LIN {X 0,Y 467.598,Z 337.24,A -85,B 0,C 180,E1 -7780.262,E2 -7780.262} C_VEL
LIN {X 0,Y 467.588,Z 337.241,A -85,B 0,C 180,E1 -7782.567,E2 -7782.567} C_VEL
LIN {X 0,Y 467.573,Z 337.242,A -85,B 0,C 180,E1 -7785.053,E2 -7785.053} C_VEL
LIN {X 0,Y 467.59,Z 337.241,A -85,B 0,C 180,E1 -7787.44,E2 -7787.44} C_VEL
LIN {X 0,Y 467.584,Z 337.244,A -85,B 0,C 180,E1 -7790.855,E2 -7790.855} C_VEL
LIN {X 0,Y 467.561,Z 337.244,A -85,B 0,C 180,E1 -7794.261,E2 -7794.261} C_VEL
LIN {X 0,Y 467.583,Z 337.239,A -85,B 0,C 180,E1 -7797.321,E2 -7797.321} C_VEL
LIN {X 0,Y 467.571,Z 337.241,A -85,B 0,C 180,E1 -7800.667,E2 -7800.667} C_VEL
LIN {X 0,Y 467.618,Z 337.238,A -85,B 0,C 180,E1 -7803.2,E2 -7803.2} C_VEL
LIN {X 0,Y 467.594,Z 337.24,A -85,B 0,C 180,E1 -7806.468,E2 -7806.468} C_VEL
LIN {X 0,Y 467.625,Z 337.233,A -85,B 0,C 180,E1 -7809.777,E2 -7809.777} C_VEL
LIN {X 0,Y 467.591,Z 337.238,A -85,B 0,C 180,E1 -7812.902,E2 -7812.902} C_VEL
LIN {X 0,Y 466.915,Z 337.324,A -85,B 0,C 180,E1 -7813.621,E2 -7813.621} C_VEL
LIN {X 0,Y 464.043,Z 337.68,A -85,B 0,C 180,E1 -7814.788,E2 -7814.788} C_VEL
LIN {X 0,Y 461.631,Z 337.984,A -85,B 0,C 180,E1 -7815.729,E2 -7815.729} C_VEL
LIN {X 0,Y 460.615,Z 338.108,A -85,B 0,C 180,E1 -7816.456,E2 -7816.456} C_VEL
LIN {X 0,Y 460.543,Z 338.117,A -85,B 0,C 180,E1 -7816.703,E2 -7816.703} C_VEL
LIN {X 0,Y 460.581,Z 338.114,A -85,B 0,C 180,E1 -7819.449,E2 -7819.449} C_VEL
LIN {X 0,Y 460.716,Z 338.099,A -85,B 0,C 180,E1 -7822.543,E2 -7822.543} C_VEL
LIN {X 0,Y 460.697,Z 338.099,A -85,B 0,C 180,E1 -7824.748,E2 -7824.748} C_VEL
LIN {X 0,Y 460.826,Z 338.08,A -85,B 0,C 180,E1 -7827.378,E2 -7827.378} C_VEL
LIN {X 0,Y 460.854,Z 338.082,A -85,B 0,C 180,E1 -7830,E2 -7830} C_VEL
LIN {X 0,Y 460.827,Z 338.081,A -85,B 0,C 180,E1 -7832.622,E2 -7832.622} C_VEL
LIN {X 0,Y 460.704,Z 338.097,A -85,B 0,C 180,E1 -7836.13,E2 -7836.13} C_VEL
LIN {X 0,Y 460.631,Z 338.108,A -85,B 0,C 180,E1 -7838.776,E2 -7838.776} C_VEL
LIN {X 0,Y 460.615,Z 338.109,A -85,B 0,C 180,E1 -7842.445,E2 -7842.445} C_VEL
LIN {X 0,Y 460.601,Z 338.111,A -85,B 0,C 180,E1 -7845.998,E2 -7845.998} C_VEL
LIN {X 0,Y 460.573,Z 338.113,A -85,B 0,C 180,E1 -7848.902,E2 -7848.902} C_VEL
LIN {X 0,Y 460.517,Z 338.122,A -85,B 0,C 180,E1 -7851.486,E2 -7851.486} C_VEL
LIN {X 0,Y 460.543,Z 338.119,A -85,B 0,C 180,E1 -7854.332,E2 -7854.332} C_VEL
LIN {X 0,Y 460.575,Z 338.113,A -85,B 0,C 180,E1 -7857.244,E2 -7857.244} C_VEL
LIN {X 0,Y 460.512,Z 338.121,A -85,B 0,C 180,E1 -7860.24,E2 -7860.24} C_VEL
LIN {X 0,Y 460.531,Z 338.121,A -85,B 0,C 180,E1 -7863.325,E2 -7863.325} C_VEL
LIN {X 0,Y 460.478,Z 338.124,A -85,B 0,C 180,E1 -7866.53,E2 -7866.53} C_VEL
LIN {X 0,Y 460.535,Z 338.118,A -85,B 0,C 180,E1 -7869.863,E2 -7869.863} C_VEL
LIN {X 0,Y 460.545,Z 338.118,A -85,B 0,C 180,E1 -7872.905,E2 -7872.905} C_VEL
LIN {X 0,Y 460.514,Z 338.123,A -85,B 0,C 180,E1 -7875.831,E2 -7875.831} C_VEL
LIN {X 0,Y 460.534,Z 338.119,A -85,B 0,C 180,E1 -7878.989,E2 -7878.989} C_VEL
LIN {X 0,Y 460.529,Z 338.122,A -85,B 0,C 180,E1 -7881.267,E2 -7881.267} C_VEL
LIN {X 0,Y 460.514,Z 338.121,A -85,B 0,C 180,E1 -7884.555,E2 -7884.555} C_VEL
LIN {X 0,Y 460.535,Z 338.119,A -85,B 0,C 180,E1 -7887.716,E2 -7887.716} C_VEL
LIN {X 0,Y 460.544,Z 338.117,A -85,B 0,C 180,E1 -7890.769,E2 -7890.769} C_VEL
LIN {X 0,Y 460.568,Z 338.115,A -85,B 0,C 180,E1 -7893.735,E2 -7893.735} C_VEL
LIN {X 0,Y 460.55,Z 338.116,A -85,B 0,C 180,E1 -7896.624,E2 -7896.624} C_VEL
LIN {X 0,Y 460.555,Z 338.114,A -85,B 0,C 180,E1 -7899.453,E2 -7899.453} C_VEL
LIN {X 0,Y 460.562,Z 338.115,A -85,B 0,C 180,E1 -7902.23,E2 -7902.23} C_VEL
LIN {X 0,Y 460.571,Z 338.114,A -85,B 0,C 180,E1 -7904.965,E2 -7904.965} C_VEL
LIN {X 0,Y 460.617,Z 338.108,A -85,B 0,C 180,E1 -7908.56,E2 -7908.56} C_VEL
LIN {X 0,Y 460.701,Z 338.097,A -85,B 0,C 180,E1 -7912.109,E2 -7912.109} C_VEL
LIN {X 0,Y 460.701,Z 338.102,A -85,B 0,C 180,E1 -7914.748,E2 -7914.748} C_VEL
LIN {X 0,Y 460.804,Z 338.082,A -85,B 0,C 180,E1 -7917.378,E2 -7917.378} C_VEL
LIN {X 0,Y 460.859,Z 338.079,A -85,B 0,C 180,E1 -7920,E2 -7920} C_VEL
LIN {X 0,Y 460.83,Z 338.081,A -85,B 0,C 180,E1 -7922.622,E2 -7922.622} C_VEL
LIN {X 0,Y 460.705,Z 338.098,A -85,B 0,C 180,E1 -7926.13,E2 -7926.13} C_VEL
LIN {X 0,Y 460.625,Z 338.11,A -85,B 0,C 180,E1 -7928.776,E2 -7928.776} C_VEL
LIN {X 0,Y 460.619,Z 338.112,A -85,B 0,C 180,E1 -7932.445,E2 -7932.445} C_VEL
LIN {X 0,Y 460.606,Z 338.112,A -85,B 0,C 180,E1 -7935.998,E2 -7935.998} C_VEL
LIN {X 0,Y 460.577,Z 338.112,A -85,B 0,C 180,E1 -7938.902,E2 -7938.902} C_VEL
LIN {X 0,Y 460.521,Z 338.122,A -85,B 0,C 180,E1 -7941.486,E2 -7941.486} C_VEL
LIN {X 0,Y 460.547,Z 338.117,A -85,B 0,C 180,E1 -7944.332,E2 -7944.332} C_VEL
LIN {X 0,Y 460.578,Z 338.113,A -85,B 0,C 180,E1 -7947.244,E2 -7947.244} C_VEL
LIN {X 0,Y 460.516,Z 338.124,A -85,B 0,C 180,E1 -7950.24,E2 -7950.24} C_VEL
LIN {X 0,Y 460.534,Z 338.117,A -85,B 0,C 180,E1 -7953.325,E2 -7953.325} C_VEL
LIN {X 0,Y 460.483,Z 338.124,A -85,B 0,C 180,E1 -7956.529,E2 -7956.529} C_VEL
LIN {X 0,Y 460.55,Z 338.117,A -85,B 0,C 180,E1 -7958.898,E2 -7958.898} C_VEL
LIN {X 0,Y 460.527,Z 338.121,A -85,B 0,C 180,E1 -7962.181,E2 -7962.181} C_VEL
LIN {X 0,Y 460.525,Z 338.12,A -85,B 0,C 180,E1 -7965.412,E2 -7965.412} C_VEL
LIN {X 0,Y 460.571,Z 338.31,A -85,B 0,C 180,E1 -7968.756,E2 -7968.756} C_VEL
LIN {X 0,Y 462.718,Z 348.896,A -85,B 0,C 180,E1 -7971.857,E2 -7971.857} C_VEL
LIN {X 0,Y 463.646,Z 354.59,A -85,B 0,C 180,E1 -7973.454,E2 -7973.454} C_VEL
LIN {X 0,Y 463.132,Z 363.771,A -85,B 0,C 180,E1 -7975.842,E2 -7975.842} C_VEL
LIN {X 0,Y 462.412,Z 376.769,A -85,B 0,C 180,E1 -7979.139,E2 -7979.139} C_VEL
LIN {X 0,Y 461.808,Z 389.925,A -85,B 0,C 180,E1 -7982.39,E2 -7982.39} C_VEL
LIN {X 0,Y 461.251,Z 403.652,A -85,B 0,C 180,E1 -7985.707,E2 -7985.707} C_VEL
LIN {X 0,Y 460.785,Z 417.545,A -85,B 0,C 180,E1 -7988.996,E2 -7988.996} C_VEL
LIN {X 0,Y 460.418,Z 431.373,A -85,B 0,C 180,E1 -7992.224,E2 -7992.224} C_VEL
LIN {X 0,Y 460.213,Z 440.731,A -85,B 0,C 180,E1 -7994.39,E2 -7994.39} C_VEL
LIN {X 0,Y 461.598,Z 455.243,A -85,B 0,C 180,E1 -7994.821,E2 -7994.821} C_VEL
LIN {X 0,Y 462.615,Z 466.865,A -85,B 0,C 180,E1 -7995.314,E2 -7995.314} C_VEL
LIN {X 0,Y 462.114,Z 478.343,A -85,B 0,C 180,E1 -7995.916,E2 -7995.916} C_VEL
LIN {X 0,Y 461.604,Z 489.684,A -85,B 0,C 180,E1 -7996.686,E2 -7996.686} C_VEL
LIN {X 0,Y 461.147,Z 501.298,A -85,B 0,C 180,E1 -7997.68,E2 -7997.68} C_VEL
LIN {X 0,Y 460.644,Z 511.654,A -85,B 0,C 180,E1 -7998.783,E2 -7998.783} C_VEL
LIN {X 0,Y 460.277,Z 520.097,A -85,B 0,C 180,E1 -7999.887,E2 -7999.887} C_VEL
LIN {X 0,Y 460.023,Z 528.384,A -85,B 0,C 180,E1 -8001.212,E2 -8001.212} C_VEL
LIN {X 0,Y 459.932,Z 535.07,A -85,B 0,C 180,E1 -8002.537,E2 -8002.537} C_VEL
LIN {X 0,Y 459.913,Z 540.386,A -85,B 0,C 180,E1 -8003.859,E2 -8003.859} C_VEL
LIN {X 0,Y 459.893,Z 544.486,A -85,B 0,C 180,E1 -8005.179,E2 -8005.179} C_VEL
LIN {X 0,Y 459.918,Z 547.493,A -85,B 0,C 180,E1 -8006.496,E2 -8006.496} C_VEL
LIN {X 0,Y 459.904,Z 548.924,A -85,B 0,C 180,E1 -8007.372,E2 -8007.372} C_VEL
LIN {X 0,Y 459.897,Z 549.91,A -85,B 0,C 180,E1 -8008.249,E2 -8008.249} C_VEL
LIN {X 0,Y 460.04,Z 550.668,A -85,B 0,C 180,E1 -8010,E2 -8010} C_VEL
LIN {X 0,Y 460.058,Z 550.379,A -85,B 0,C 180,E1 -8010.875,E2 -8010.875} C_VEL
LIN {X 0,Y 459.953,Z 548.51,A -85,B 0,C 180,E1 -8012.627,E2 -8012.627} C_VEL
LIN {X 0,Y 460.005,Z 545.972,A -85,B 0,C 180,E1 -8013.942,E2 -8013.942} C_VEL
LIN {X 0,Y 459.99,Z 542.372,A -85,B 0,C 180,E1 -8015.26,E2 -8015.26} C_VEL
LIN {X 0,Y 459.99,Z 537.034,A -85,B 0,C 180,E1 -8016.729,E2 -8016.729} C_VEL
LIN {X 0,Y 460.043,Z 530.486,A -85,B 0,C 180,E1 -8018.124,E2 -8018.124} C_VEL
LIN {X 0,Y 460.195,Z 522.709,A -85,B 0,C 180,E1 -8019.449,E2 -8019.449} C_VEL
LIN {X 0,Y 460.5,Z 513.145,A -85,B 0,C 180,E1 -8020.775,E2 -8020.775} C_VEL
LIN {X 0,Y 460.903,Z 503.312,A -85,B 0,C 180,E1 -8021.879,E2 -8021.879} C_VEL
LIN {X 0,Y 461.223,Z 493.086,A -85,B 0,C 180,E1 -8022.826,E2 -8022.826} C_VEL
LIN {X 0,Y 461.773,Z 480.667,A -85,B 0,C 180,E1 -8023.757,E2 -8023.757} C_VEL
LIN {X 0,Y 462.365,Z 467.344,A -85,B 0,C 180,E1 -8024.525,E2 -8024.525} C_VEL
LIN {X 0,Y 461.97,Z 461.418,A -85,B 0,C 180,E1 -8024.819,E2 -8024.819} C_VEL
LIN {X 0,Y 461.138,Z 447.636,A -85,B 0,C 180,E1 -8025.371,E2 -8025.371} C_VEL
LIN {X 0,Y 460.184,Z 436.063,A -85,B 0,C 180,E1 -8025.707,E2 -8025.707} C_VEL
LIN {X 0,Y 460.345,Z 423.4,A -85,B 0,C 180,E1 -8028.469,E2 -8028.469} C_VEL
LIN {X 0,Y 460.504,Z 409.727,A -85,B 0,C 180,E1 -8031.486,E2 -8031.486} C_VEL
LIN {X 0,Y 460.723,Z 396.07,A -85,B 0,C 180,E1 -8034.562,E2 -8034.562} C_VEL
LIN {X 0,Y 461.007,Z 383.272,A -85,B 0,C 180,E1 -8037.534,E2 -8037.534} C_VEL
LIN {X 0,Y 461.36,Z 370.292,A -85,B 0,C 180,E1 -8040.685,E2 -8040.685} C_VEL
LIN {X 0,Y 461.759,Z 360.404,A -85,B 0,C 180,E1 -8043.225,E2 -8043.225} C_VEL
LIN {X 0,Y 462.522,Z 350.975,A -85,B 0,C 180,E1 -8045.804,E2 -8045.804} C_VEL
LIN {X 0,Y 462.353,Z 347.344,A -85,B 0,C 180,E1 -8046.9,E2 -8046.9} C_VEL
LIN {X 0,Y 460.967,Z 340.192,A -85,B 0,C 180,E1 -8049.354,E2 -8049.354} C_VEL
LIN {X 0,Y 460.548,Z 338.121,A -85,B 0,C 180,E1 -8050.196,E2 -8050.196} C_VEL
LIN {X 0,Y 460.504,Z 338.125,A -85,B 0,C 180,E1 -8053.375,E2 -8053.375} C_VEL
LIN {X 0,Y 460.504,Z 338.123,A -85,B 0,C 180,E1 -8056.625,E2 -8056.625} C_VEL
LIN {X 0,Y 460.545,Z 338.118,A -85,B 0,C 180,E1 -8059.731,E2 -8059.731} C_VEL
LIN {X 0,Y 460.531,Z 338.119,A -85,B 0,C 180,E1 -8062.519,E2 -8062.519} C_VEL
LIN {X 0,Y 460.552,Z 338.118,A -85,B 0,C 180,E1 -8065.624,E2 -8065.624} C_VEL
LIN {X 0,Y 460.541,Z 338.118,A -85,B 0,C 180,E1 -8068.745,E2 -8068.745} C_VEL
LIN {X 0,Y 460.586,Z 338.112,A -85,B 0,C 180,E1 -8072.254,E2 -8072.254} C_VEL
LIN {X 0,Y 460.544,Z 338.118,A -85,B 0,C 180,E1 -8074.704,E2 -8074.704} C_VEL
LIN {X 0,Y 460.515,Z 338.123,A -85,B 0,C 180,E1 -8077.571,E2 -8077.571} C_VEL
LIN {X 0,Y 460.573,Z 338.117,A -85,B 0,C 180,E1 -8080.385,E2 -8080.385} C_VEL
LIN {X 0,Y 460.569,Z 338.116,A -85,B 0,C 180,E1 -8083.146,E2 -8083.146} C_VEL
LIN {X 0,Y 460.633,Z 338.213,A -85,B 0,C 180,E1 -8084.134,E2 -8084.134} C_VEL
LIN {X 0,Y 463.679,Z 348.826,A -85,B 0,C 180,E1 -8084.843,E2 -8084.843} C_VEL
LIN {X 0,Y 463.301,Z 360.273,A -85,B 0,C 180,E1 -8085.617,E2 -8085.617} C_VEL
LIN {X 0,Y 462.89,Z 371.591,A -85,B 0,C 180,E1 -8086.594,E2 -8086.594} C_VEL
LIN {X 0,Y 462.45,Z 380.084,A -85,B 0,C 180,E1 -8087.493,E2 -8087.493} C_VEL
LIN {X 0,Y 461.951,Z 388.673,A -85,B 0,C 180,E1 -8088.593,E2 -8088.593} C_VEL
LIN {X 0,Y 461.543,Z 397.068,A -85,B 0,C 180,E1 -8089.915,E2 -8089.915} C_VEL
LIN {X 0,Y 461.19,Z 403.729,A -85,B 0,C 180,E1 -8091.234,E2 -8091.234} C_VEL
LIN {X 0,Y 460.817,Z 409.881,A -85,B 0,C 180,E1 -8092.801,E2 -8092.801} C_VEL
LIN {X 0,Y 460.572,Z 414.264,A -85,B 0,C 180,E1 -8094.308,E2 -8094.308} C_VEL
LIN {X 0,Y 460.387,Z 416.971,A -85,B 0,C 180,E1 -8095.622,E2 -8095.622} C_VEL
LIN {X 0,Y 460.314,Z 418.215,A -85,B 0,C 180,E1 -8096.499,E2 -8096.499} C_VEL
LIN {X 0,Y 460.232,Z 419.525,A -85,B 0,C 180,E1 -8098.25,E2 -8098.25} C_VEL
LIN {X 0,Y 460.185,Z 419.587,A -85,B 0,C 180,E1 -8099.125,E2 -8099.125} C_VEL
LIN {X 0,Y 460.162,Z 418.481,A -85,B 0,C 180,E1 -8100.875,E2 -8100.875} C_VEL
LIN {X 0,Y 460.236,Z 417.34,A -85,B 0,C 180,E1 -8101.75,E2 -8101.75} C_VEL
LIN {X 0,Y 460.28,Z 414.837,A -85,B 0,C 180,E1 -8103.063,E2 -8103.063} C_VEL
LIN {X 0,Y 460.423,Z 411.338,A -85,B 0,C 180,E1 -8104.377,E2 -8104.377} C_VEL
LIN {X 0,Y 460.603,Z 406.758,A -85,B 0,C 180,E1 -8105.692,E2 -8105.692} C_VEL
LIN {X 0,Y 461.037,Z 399.83,A -85,B 0,C 180,E1 -8107.222,E2 -8107.222} C_VEL
LIN {X 0,Y 461.343,Z 392.328,A -85,B 0,C 180,E1 -8108.542,E2 -8108.542} C_VEL
LIN {X 0,Y 461.654,Z 384.704,A -85,B 0,C 180,E1 -8109.64,E2 -8109.64} C_VEL
LIN {X 0,Y 462.091,Z 375.474,A -85,B 0,C 180,E1 -8110.738,E2 -8110.738} C_VEL
LIN {X 0,Y 462.52,Z 365.237,A -85,B 0,C 180,E1 -8111.726,E2 -8111.726} C_VEL
LIN {X 0,Y 462.763,Z 356.364,A -85,B 0,C 180,E1 -8112.439,E2 -8112.439} C_VEL
LIN {X 0,Y 463.121,Z 347.588,A -85,B 0,C 180,E1 -8113.023,E2 -8113.023} C_VEL
LIN {X 0,Y 460.601,Z 338.114,A -85,B 0,C 180,E1 -8113.635,E2 -8113.635} C_VEL
LIN {X 0,Y 460.562,Z 338.114,A -85,B 0,C 180,E1 -8116.854,E2 -8116.854} C_VEL
LIN {X 0,Y 460.571,Z 338.113,A -85,B 0,C 180,E1 -8119.615,E2 -8119.615} C_VEL
LIN {X 0,Y 460.515,Z 338.121,A -85,B 0,C 180,E1 -8122.428,E2 -8122.428} C_VEL
LIN {X 0,Y 460.571,Z 338.115,A -85,B 0,C 180,E1 -8125.802,E2 -8125.802} C_VEL
LIN {X 0,Y 460.559,Z 338.117,A -85,B 0,C 180,E1 -8128.232,E2 -8128.232} C_VEL
LIN {X 0,Y 460.525,Z 338.123,A -85,B 0,C 180,E1 -8131.283,E2 -8131.283} C_VEL
LIN {X 0,Y 460.535,Z 338.118,A -85,B 0,C 180,E1 -8134.505,E2 -8134.505} C_VEL
LIN {X 0,Y 460.531,Z 338.117,A -85,B 0,C 180,E1 -8137.62,E2 -8137.62} C_VEL
LIN {X 0,Y 460.561,Z 338.117,A -85,B 0,C 180,E1 -8140.272,E2 -8140.272} C_VEL
LIN {X 0,Y 460.502,Z 338.124,A -85,B 0,C 180,E1 -8143.375,E2 -8143.375} C_VEL
LIN {X 0,Y 460.515,Z 338.121,A -85,B 0,C 180,E1 -8146.626,E2 -8146.626} C_VEL
LIN {X 0,Y 460.544,Z 338.117,A -85,B 0,C 180,E1 -8149.73,E2 -8149.73} C_VEL
LIN {X 0,Y 460.501,Z 338.125,A -85,B 0,C 180,E1 -8152.524,E2 -8152.524} C_VEL
LIN {X 0,Y 460.547,Z 338.115,A -85,B 0,C 180,E1 -8155.624,E2 -8155.624} C_VEL
LIN {X 0,Y 460.538,Z 338.118,A -85,B 0,C 180,E1 -8158.744,E2 -8158.744} C_VEL
LIN {X 0,Y 460.59,Z 338.112,A -85,B 0,C 180,E1 -8162.252,E2 -8162.252} C_VEL
LIN {X 0,Y 460.56,Z 338.117,A -85,B 0,C 180,E1 -8164.705,E2 -8164.705} C_VEL
LIN {X 0,Y 460.513,Z 338.12,A -85,B 0,C 180,E1 -8167.571,E2 -8167.571} C_VEL
LIN {X 0,Y 460.571,Z 338.118,A -85,B 0,C 180,E1 -8170.384,E2 -8170.384} C_VEL
LIN {X 0,Y 460.567,Z 338.112,A -85,B 0,C 180,E1 -8173.146,E2 -8173.146} C_VEL
LIN {X 0,Y 460.557,Z 338.119,A -85,B 0,C 180,E1 -8175.868,E2 -8175.868} C_VEL
LIN {X 0,Y 460.543,Z 338.117,A -85,B 0,C 180,E1 -8176.703,E2 -8176.703} C_VEL
LIN {X 0,Y 459.907,Z 338.198,A -85,B 0,C 180,E1 -8177.433,E2 -8177.433} C_VEL
LIN {X 0,Y 457.078,Z 338.55,A -85,B 0,C 180,E1 -8178.62,E2 -8178.62} C_VEL
LIN {X 0,Y 454.674,Z 338.851,A -85,B 0,C 180,E1 -8179.576,E2 -8179.576} C_VEL
LIN {X 0,Y 453.648,Z 338.976,A -85,B 0,C 180,E1 -8180.316,E2 -8180.316} C_VEL
LIN {X 0,Y 453.569,Z 338.985,A -85,B 0,C 180,E1 -8180.566,E2 -8180.566} C_VEL
LIN {X 0,Y 453.631,Z 338.979,A -85,B 0,C 180,E1 -8182.88,E2 -8182.88} C_VEL
LIN {X 0,Y 453.67,Z 338.975,A -85,B 0,C 180,E1 -8184.667,E2 -8184.667} C_VEL
LIN {X 0,Y 453.766,Z 338.96,A -85,B 0,C 180,E1 -8187.337,E2 -8187.337} C_VEL
LIN {X 0,Y 453.824,Z 338.958,A -85,B 0,C 180,E1 -8190,E2 -8190} C_VEL
LIN {X 0,Y 453.767,Z 338.96,A -85,B 0,C 180,E1 -8192.663,E2 -8192.663} C_VEL
LIN {X 0,Y 453.671,Z 338.973,A -85,B 0,C 180,E1 -8196.225,E2 -8196.225} C_VEL
LIN {X 0,Y 453.594,Z 338.984,A -85,B 0,C 180,E1 -8198.913,E2 -8198.913} C_VEL
LIN {X 0,Y 453.565,Z 338.987,A -85,B 0,C 180,E1 -8202.529,E2 -8202.529} C_VEL
LIN {X 0,Y 453.546,Z 338.988,A -85,B 0,C 180,E1 -8206.196,E2 -8206.196} C_VEL
LIN {X 0,Y 453.522,Z 338.991,A -85,B 0,C 180,E1 -8209.041,E2 -8209.041} C_VEL
LIN {X 0,Y 453.478,Z 338.997,A -85,B 0,C 180,E1 -8211.836,E2 -8211.836} C_VEL
LIN {X 0,Y 453.515,Z 338.994,A -85,B 0,C 180,E1 -8214.735,E2 -8214.735} C_VEL
LIN {X 0,Y 453.534,Z 338.994,A -85,B 0,C 180,E1 -8217.96,E2 -8217.96} C_VEL
LIN {X 0,Y 453.468,Z 339.001,A -85,B 0,C 180,E1 -8221.526,E2 -8221.526} C_VEL
LIN {X 0,Y 453.489,Z 338.994,A -85,B 0,C 180,E1 -8224.778,E2 -8224.778} C_VEL
LIN {X 0,Y 453.467,Z 338.999,A -85,B 0,C 180,E1 -8228.312,E2 -8228.312} C_VEL
LIN {X 0,Y 453.497,Z 338.996,A -85,B 0,C 180,E1 -8230.609,E2 -8230.609} C_VEL
LIN {X 0,Y 453.485,Z 338.997,A -85,B 0,C 180,E1 -8233.248,E2 -8233.248} C_VEL
LIN {X 0,Y 453.469,Z 339.001,A -85,B 0,C 180,E1 -8235.779,E2 -8235.779} C_VEL
LIN {X 0,Y 453.482,Z 338.996,A -85,B 0,C 180,E1 -8238.21,E2 -8238.21} C_VEL
LIN {X 0,Y 453.497,Z 338.995,A -85,B 0,C 180,E1 -8240.794,E2 -8240.794} C_VEL
LIN {X 0,Y 453.458,Z 338.998,A -85,B 0,C 180,E1 -8243.918,E2 -8243.918} C_VEL
LIN {X 0,Y 453.486,Z 338.997,A -85,B 0,C 180,E1 -8247.152,E2 -8247.152} C_VEL
LIN {X 0,Y 453.479,Z 338.999,A -85,B 0,C 180,E1 -8250.269,E2 -8250.269} C_VEL
LIN {X 0,Y 453.514,Z 338.996,A -85,B 0,C 180,E1 -8253.295,E2 -8253.295} C_VEL
LIN {X 0,Y 453.507,Z 338.993,A -85,B 0,C 180,E1 -8256.239,E2 -8256.239} C_VEL
LIN {X 0,Y 453.487,Z 338.997,A -85,B 0,C 180,E1 -8259.118,E2 -8259.118} C_VEL
LIN {X 0,Y 453.515,Z 338.992,A -85,B 0,C 180,E1 -8261.945,E2 -8261.945} C_VEL
LIN {X 0,Y 453.545,Z 338.99,A -85,B 0,C 180,E1 -8264.727,E2 -8264.727} C_VEL
LIN {X 0,Y 453.565,Z 338.987,A -85,B 0,C 180,E1 -8268.379,E2 -8268.379} C_VEL
LIN {X 0,Y 453.658,Z 338.975,A -85,B 0,C 180,E1 -8271.985,E2 -8271.985} C_VEL
LIN {X 0,Y 453.675,Z 338.976,A -85,B 0,C 180,E1 -8274.667,E2 -8274.667} C_VEL
LIN {X 0,Y 453.748,Z 338.961,A -85,B 0,C 180,E1 -8277.337,E2 -8277.337} C_VEL
LIN {X 0,Y 453.829,Z 338.954,A -85,B 0,C 180,E1 -8280,E2 -8280} C_VEL
LIN {X 0,Y 453.77,Z 338.961,A -85,B 0,C 180,E1 -8282.663,E2 -8282.663} C_VEL
LIN {X 0,Y 453.672,Z 338.973,A -85,B 0,C 180,E1 -8286.226,E2 -8286.226} C_VEL
LIN {X 0,Y 453.591,Z 338.985,A -85,B 0,C 180,E1 -8288.914,E2 -8288.914} C_VEL
LIN {X 0,Y 453.569,Z 338.989,A -85,B 0,C 180,E1 -8292.529,E2 -8292.529} C_VEL
LIN {X 0,Y 453.55,Z 338.992,A -85,B 0,C 180,E1 -8296.196,E2 -8296.196} C_VEL
LIN {X 0,Y 453.527,Z 338.991,A -85,B 0,C 180,E1 -8299.041,E2 -8299.041} C_VEL
LIN {X 0,Y 453.482,Z 338.999,A -85,B 0,C 180,E1 -8301.836,E2 -8301.836} C_VEL
LIN {X 0,Y 453.519,Z 338.994,A -85,B 0,C 180,E1 -8304.734,E2 -8304.734} C_VEL
LIN {X 0,Y 453.537,Z 338.991,A -85,B 0,C 180,E1 -8307.96,E2 -8307.96} C_VEL
LIN {X 0,Y 453.471,Z 338.997,A -85,B 0,C 180,E1 -8311.525,E2 -8311.525} C_VEL
LIN {X 0,Y 453.494,Z 338.994,A -85,B 0,C 180,E1 -8314.777,E2 -8314.777} C_VEL
LIN {X 0,Y 453.478,Z 338.997,A -85,B 0,C 180,E1 -8318.311,E2 -8318.311} C_VEL
LIN {X 0,Y 453.498,Z 338.996,A -85,B 0,C 180,E1 -8320.609,E2 -8320.609} C_VEL
LIN {X 0,Y 453.46,Z 339,A -85,B 0,C 180,E1 -8323.244,E2 -8323.244} C_VEL
LIN {X 0,Y 453.478,Z 339,A -85,B 0,C 180,E1 -8325.78,E2 -8325.78} C_VEL
LIN {X 0,Y 453.527,Z 339.118,A -85,B 0,C 180,E1 -8328.447,E2 -8328.447} C_VEL
LIN {X 0,Y 455.452,Z 348.745,A -85,B 0,C 180,E1 -8331.322,E2 -8331.322} C_VEL
LIN {X 0,Y 456.645,Z 355.141,A -85,B 0,C 180,E1 -8333.16,E2 -8333.16} C_VEL
LIN {X 0,Y 456.403,Z 361.922,A -85,B 0,C 180,E1 -8334.976,E2 -8334.976} C_VEL
LIN {X 0,Y 455.579,Z 375.018,A -85,B 0,C 180,E1 -8338.365,E2 -8338.365} C_VEL
LIN {X 0,Y 454.839,Z 389.623,A -85,B 0,C 180,E1 -8342.05,E2 -8342.05} C_VEL
LIN {X 0,Y 454.26,Z 402.862,A -85,B 0,C 180,E1 -8345.309,E2 -8345.309} C_VEL
LIN {X 0,Y 453.8,Z 415.29,A -85,B 0,C 180,E1 -8348.314,E2 -8348.314} C_VEL
LIN {X 0,Y 453.368,Z 430.488,A -85,B 0,C 180,E1 -8351.938,E2 -8351.938} C_VEL
LIN {X 0,Y 453.118,Z 439.854,A -85,B 0,C 180,E1 -8354.146,E2 -8354.146} C_VEL
LIN {X 0,Y 454.661,Z 455.955,A -85,B 0,C 180,E1 -8354.659,E2 -8354.659} C_VEL
LIN {X 0,Y 455.597,Z 467.856,A -85,B 0,C 180,E1 -8355.197,E2 -8355.197} C_VEL
LIN {X 0,Y 455.013,Z 480.558,A -85,B 0,C 180,E1 -8355.92,E2 -8355.92} C_VEL
LIN {X 0,Y 454.424,Z 492.213,A -85,B 0,C 180,E1 -8356.775,E2 -8356.775} C_VEL
LIN {X 0,Y 454.01,Z 503.472,A -85,B 0,C 180,E1 -8357.824,E2 -8357.824} C_VEL
LIN {X 0,Y 453.54,Z 512.327,A -85,B 0,C 180,E1 -8358.831,E2 -8358.831} C_VEL
LIN {X 0,Y 453.091,Z 521.996,A -85,B 0,C 180,E1 -8360.176,E2 -8360.176} C_VEL
LIN {X 0,Y 452.948,Z 529.726,A -85,B 0,C 180,E1 -8361.523,E2 -8361.523} C_VEL
LIN {X 0,Y 452.84,Z 535.933,A -85,B 0,C 180,E1 -8362.868,E2 -8362.868} C_VEL
LIN {X 0,Y 452.834,Z 540.842,A -85,B 0,C 180,E1 -8364.21,E2 -8364.21} C_VEL
LIN {X 0,Y 452.857,Z 544.583,A -85,B 0,C 180,E1 -8365.549,E2 -8365.549} C_VEL
LIN {X 0,Y 452.874,Z 546.492,A -85,B 0,C 180,E1 -8366.441,E2 -8366.441} C_VEL
LIN {X 0,Y 452.86,Z 547.93,A -85,B 0,C 180,E1 -8367.331,E2 -8367.331} C_VEL
LIN {X 0,Y 452.86,Z 548.914,A -85,B 0,C 180,E1 -8368.221,E2 -8368.221} C_VEL
LIN {X 0,Y 453.019,Z 549.668,A -85,B 0,C 180,E1 -8370,E2 -8370} C_VEL
LIN {X 0,Y 453.038,Z 549.375,A -85,B 0,C 180,E1 -8370.889,E2 -8370.889} C_VEL
LIN {X 0,Y 452.913,Z 547.486,A -85,B 0,C 180,E1 -8372.668,E2 -8372.668} C_VEL
LIN {X 0,Y 452.964,Z 544.932,A -85,B 0,C 180,E1 -8374.004,E2 -8374.004} C_VEL
LIN {X 0,Y 452.919,Z 541.304,A -85,B 0,C 180,E1 -8375.342,E2 -8375.342} C_VEL
LIN {X 0,Y 452.93,Z 536.296,A -85,B 0,C 180,E1 -8376.746,E2 -8376.746} C_VEL
LIN {X 0,Y 453.007,Z 529.387,A -85,B 0,C 180,E1 -8378.251,E2 -8378.251} C_VEL
LIN {X 0,Y 453.129,Z 521.592,A -85,B 0,C 180,E1 -8379.598,E2 -8379.598} C_VEL
LIN {X 0,Y 453.449,Z 512.01,A -85,B 0,C 180,E1 -8380.945,E2 -8380.945} C_VEL
LIN {X 0,Y 453.923,Z 502.2,A -85,B 0,C 180,E1 -8382.065,E2 -8382.065} C_VEL
LIN {X 0,Y 454.222,Z 492.333,A -85,B 0,C 180,E1 -8382.998,E2 -8382.998} C_VEL
LIN {X 0,Y 454.819,Z 479.625,A -85,B 0,C 180,E1 -8383.972,E2 -8383.972} C_VEL
LIN {X 0,Y 455.459,Z 466.458,A -85,B 0,C 180,E1 -8384.75,E2 -8384.75} C_VEL
LIN {X 0,Y 454.574,Z 454.717,A -85,B 0,C 180,E1 -8385.322,E2 -8385.322} C_VEL
LIN {X 0,Y 453.76,Z 441.225,A -85,B 0,C 180,E1 -8385.81,E2 -8385.81} C_VEL
LIN {X 0,Y 453.114,Z 434.683,A -85,B 0,C 180,E1 -8386.008,E2 -8386.008} C_VEL
LIN {X 0,Y 453.257,Z 421.226,A -85,B 0,C 180,E1 -8389.003,E2 -8389.003} C_VEL
LIN {X 0,Y 453.461,Z 407.61,A -85,B 0,C 180,E1 -8392.076,E2 -8392.076} C_VEL
LIN {X 0,Y 453.739,Z 394.043,A -85,B 0,C 180,E1 -8395.211,E2 -8395.211} C_VEL
LIN {X 0,Y 454.057,Z 381.022,A -85,B 0,C 180,E1 -8398.326,E2 -8398.326} C_VEL
LIN {X 0,Y 454.551,Z 367.463,A -85,B 0,C 180,E1 -8401.747,E2 -8401.747} C_VEL
LIN {X 0,Y 455.471,Z 353.929,A -85,B 0,C 180,E1 -8405.442,E2 -8405.442} C_VEL
LIN {X 0,Y 455.559,Z 349.88,A -85,B 0,C 180,E1 -8406.658,E2 -8406.658} C_VEL
LIN {X 0,Y 454.156,Z 342.237,A -85,B 0,C 180,E1 -8409.308,E2 -8409.308} C_VEL
LIN {X 0,Y 453.497,Z 338.999,A -85,B 0,C 180,E1 -8410.609,E2 -8410.609} C_VEL
LIN {X 0,Y 453.459,Z 339.002,A -85,B 0,C 180,E1 -8413.244,E2 -8413.244} C_VEL
LIN {X 0,Y 453.47,Z 339.001,A -85,B 0,C 180,E1 -8415.779,E2 -8415.779} C_VEL
LIN {X 0,Y 453.483,Z 338.998,A -85,B 0,C 180,E1 -8418.209,E2 -8418.209} C_VEL
LIN {X 0,Y 453.498,Z 338.995,A -85,B 0,C 180,E1 -8420.793,E2 -8420.793} C_VEL
LIN {X 0,Y 453.46,Z 339,A -85,B 0,C 180,E1 -8423.917,E2 -8423.917} C_VEL
LIN {X 0,Y 453.487,Z 338.997,A -85,B 0,C 180,E1 -8427.151,E2 -8427.151} C_VEL
LIN {X 0,Y 453.479,Z 338.997,A -85,B 0,C 180,E1 -8430.268,E2 -8430.268} C_VEL
LIN {X 0,Y 453.506,Z 338.994,A -85,B 0,C 180,E1 -8433.294,E2 -8433.294} C_VEL
LIN {X 0,Y 453.502,Z 338.996,A -85,B 0,C 180,E1 -8436.239,E2 -8436.239} C_VEL
LIN {X 0,Y 453.487,Z 338.999,A -85,B 0,C 180,E1 -8439.118,E2 -8439.118} C_VEL
LIN {X 0,Y 453.515,Z 338.995,A -85,B 0,C 180,E1 -8441.945,E2 -8441.945} C_VEL
LIN {X 0,Y 453.547,Z 338.993,A -85,B 0,C 180,E1 -8443.828,E2 -8443.828} C_VEL
LIN {X 0,Y 456.945,Z 350.447,A -85,B 0,C 180,E1 -8444.633,E2 -8444.633} C_VEL
LIN {X 0,Y 456.558,Z 361.551,A -85,B 0,C 180,E1 -8445.4,E2 -8445.4} C_VEL
LIN {X 0,Y 456.1,Z 372.644,A -85,B 0,C 180,E1 -8446.371,E2 -8446.371} C_VEL
LIN {X 0,Y 455.647,Z 381.312,A -85,B 0,C 180,E1 -8447.303,E2 -8447.303} C_VEL
LIN {X 0,Y 455.115,Z 389.886,A -85,B 0,C 180,E1 -8448.419,E2 -8448.419} C_VEL
LIN {X 0,Y 454.655,Z 398.226,A -85,B 0,C 180,E1 -8449.76,E2 -8449.76} C_VEL
LIN {X 0,Y 454.26,Z 404.85,A -85,B 0,C 180,E1 -8451.1,E2 -8451.1} C_VEL
LIN {X 0,Y 453.872,Z 410.876,A -85,B 0,C 180,E1 -8452.664,E2 -8452.664} C_VEL
LIN {X 0,Y 453.59,Z 415.347,A -85,B 0,C 180,E1 -8454.22,E2 -8454.22} C_VEL
LIN {X 0,Y 453.386,Z 418.045,A -85,B 0,C 180,E1 -8455.555,E2 -8455.555} C_VEL
LIN {X 0,Y 453.305,Z 419.284,A -85,B 0,C 180,E1 -8456.444,E2 -8456.444} C_VEL
LIN {X 0,Y 453.215,Z 420.573,A -85,B 0,C 180,E1 -8458.223,E2 -8458.223} C_VEL
LIN {X 0,Y 453.186,Z 420.619,A -85,B 0,C 180,E1 -8459.111,E2 -8459.111} C_VEL
LIN {X 0,Y 453.139,Z 419.488,A -85,B 0,C 180,E1 -8460.889,E2 -8460.889} C_VEL
LIN {X 0,Y 453.217,Z 418.329,A -85,B 0,C 180,E1 -8461.777,E2 -8461.777} C_VEL
LIN {X 0,Y 453.27,Z 415.796,A -85,B 0,C 180,E1 -8463.111,E2 -8463.111} C_VEL
LIN {X 0,Y 453.406,Z 412.266,A -85,B 0,C 180,E1 -8464.445,E2 -8464.445} C_VEL
LIN {X 0,Y 453.61,Z 407.65,A -85,B 0,C 180,E1 -8465.78,E2 -8465.78} C_VEL
LIN {X 0,Y 454.041,Z 400.685,A -85,B 0,C 180,E1 -8467.333,E2 -8467.333} C_VEL
LIN {X 0,Y 454.366,Z 393.129,A -85,B 0,C 180,E1 -8468.674,E2 -8468.674} C_VEL
LIN {X 0,Y 454.702,Z 385.458,A -85,B 0,C 180,E1 -8469.789,E2 -8469.789} C_VEL
LIN {X 0,Y 455.169,Z 376.165,A -85,B 0,C 180,E1 -8470.903,E2 -8470.903} C_VEL
LIN {X 0,Y 455.623,Z 365.87,A -85,B 0,C 180,E1 -8471.906,E2 -8471.906} C_VEL
LIN {X 0,Y 455.86,Z 357.04,A -85,B 0,C 180,E1 -8472.623,E2 -8472.623} C_VEL
LIN {X 0,Y 456.087,Z 348.491,A -85,B 0,C 180,E1 -8473.205,E2 -8473.205} C_VEL
LIN {X 0,Y 453.544,Z 338.993,A -85,B 0,C 180,E1 -8473.852,E2 -8473.852} C_VEL
LIN {X 0,Y 453.548,Z 338.987,A -85,B 0,C 180,E1 -8476.196,E2 -8476.196} C_VEL
LIN {X 0,Y 453.52,Z 338.995,A -85,B 0,C 180,E1 -8479.039,E2 -8479.039} C_VEL
LIN {X 0,Y 453.48,Z 338.996,A -85,B 0,C 180,E1 -8481.836,E2 -8481.836} C_VEL
LIN {X 0,Y 453.517,Z 338.995,A -85,B 0,C 180,E1 -8484.734,E2 -8484.734} C_VEL
LIN {X 0,Y 453.541,Z 338.99,A -85,B 0,C 180,E1 -8487.961,E2 -8487.961} C_VEL
LIN {X 0,Y 453.47,Z 339,A -85,B 0,C 180,E1 -8491.525,E2 -8491.525} C_VEL
LIN {X 0,Y 453.49,Z 338.997,A -85,B 0,C 180,E1 -8494.777,E2 -8494.777} C_VEL
LIN {X 0,Y 453.486,Z 338.996,A -85,B 0,C 180,E1 -8498.309,E2 -8498.309} C_VEL
LIN {X 0,Y 453.518,Z 338.995,A -85,B 0,C 180,E1 -8500.606,E2 -8500.606} C_VEL
LIN {X 0,Y 453.468,Z 339.001,A -85,B 0,C 180,E1 -8504.221,E2 -8504.221} C_VEL
LIN {X 0,Y 453.473,Z 339,A -85,B 0,C 180,E1 -8507.006,E2 -8507.006} C_VEL
LIN {X 0,Y 453.507,Z 338.995,A -85,B 0,C 180,E1 -8510.552,E2 -8510.552} C_VEL
LIN {X 0,Y 453.455,Z 338.998,A -85,B 0,C 180,E1 -8513.917,E2 -8513.917} C_VEL
LIN {X 0,Y 453.484,Z 338.996,A -85,B 0,C 180,E1 -8517.151,E2 -8517.151} C_VEL
LIN {X 0,Y 453.477,Z 338.999,A -85,B 0,C 180,E1 -8520.268,E2 -8520.268} C_VEL
LIN {X 0,Y 453.511,Z 338.994,A -85,B 0,C 180,E1 -8523.294,E2 -8523.294} C_VEL
LIN {X 0,Y 453.505,Z 338.994,A -85,B 0,C 180,E1 -8526.239,E2 -8526.239} C_VEL
LIN {X 0,Y 453.484,Z 338.995,A -85,B 0,C 180,E1 -8529.118,E2 -8529.118} C_VEL
LIN {X 0,Y 453.513,Z 338.993,A -85,B 0,C 180,E1 -8531.945,E2 -8531.945} C_VEL
LIN {X 0,Y 453.541,Z 338.989,A -85,B 0,C 180,E1 -8534.726,E2 -8534.726} C_VEL
LIN {X 0,Y 453.561,Z 338.987,A -85,B 0,C 180,E1 -8538.379,E2 -8538.379} C_VEL
LIN {X 0,Y 453.569,Z 338.985,A -85,B 0,C 180,E1 -8540.566,E2 -8540.566} C_VEL
LIN {X 0,Y 452.918,Z 339.068,A -85,B 0,C 180,E1 -8541.307,E2 -8541.307} C_VEL
LIN {X 0,Y 450.089,Z 339.422,A -85,B 0,C 180,E1 -8542.512,E2 -8542.512} C_VEL
LIN {X 0,Y 447.707,Z 339.716,A -85,B 0,C 180,E1 -8543.484,E2 -8543.484} C_VEL
LIN {X 0,Y 446.707,Z 339.843,A -85,B 0,C 180,E1 -8544.235,E2 -8544.235} C_VEL
LIN {X 0,Y 446.639,Z 339.85,A -85,B 0,C 180,E1 -8544.489,E2 -8544.489} C_VEL
LIN {X 0,Y 446.71,Z 339.839,A -85,B 0,C 180,E1 -8547.295,E2 -8547.295} C_VEL
LIN {X 0,Y 446.794,Z 339.833,A -85,B 0,C 180,E1 -8550,E2 -8550} C_VEL
LIN {X 0,Y 446.711,Z 339.84,A -85,B 0,C 180,E1 -8552.705,E2 -8552.705} C_VEL
LIN {X 0,Y 446.641,Z 339.85,A -85,B 0,C 180,E1 -8556.324,E2 -8556.324} C_VEL
LIN {X 0,Y 446.54,Z 339.863,A -85,B 0,C 180,E1 -8559.055,E2 -8559.055} C_VEL
LIN {X 0,Y 446.522,Z 339.863,A -85,B 0,C 180,E1 -8562.73,E2 -8562.73} C_VEL
LIN {X 0,Y 446.498,Z 339.866,A -85,B 0,C 180,E1 -8566.228,E2 -8566.228} C_VEL
LIN {X 0,Y 446.471,Z 339.872,A -85,B 0,C 180,E1 -8569.303,E2 -8569.303} C_VEL
LIN {X 0,Y 446.42,Z 339.877,A -85,B 0,C 180,E1 -8572.2,E2 -8572.2} C_VEL
LIN {X 0,Y 446.459,Z 339.873,A -85,B 0,C 180,E1 -8575.152,E2 -8575.152} C_VEL
LIN {X 0,Y 446.486,Z 339.87,A -85,B 0,C 180,E1 -8578.179,E2 -8578.179} C_VEL
LIN {X 0,Y 446.421,Z 339.879,A -85,B 0,C 180,E1 -8581.775,E2 -8581.775} C_VEL
LIN {X 0,Y 446.43,Z 339.872,A -85,B 0,C 180,E1 -8584.523,E2 -8584.523} C_VEL
LIN {X 0,Y 446.418,Z 339.876,A -85,B 0,C 180,E1 -8588.08,E2 -8588.08} C_VEL
LIN {X 0,Y 446.434,Z 339.878,A -85,B 0,C 180,E1 -8590.919,E2 -8590.919} C_VEL
LIN {X 0,Y 446.448,Z 339.875,A -85,B 0,C 180,E1 -8593.841,E2 -8593.841} C_VEL
LIN {X 0,Y 446.402,Z 339.879,A -85,B 0,C 180,E1 -8596.404,E2 -8596.404} C_VEL
LIN {X 0,Y 446.43,Z 339.877,A -85,B 0,C 180,E1 -8599.083,E2 -8599.083} C_VEL
LIN {X 0,Y 446.412,Z 339.875,A -85,B 0,C 180,E1 -8602.122,E2 -8602.122} C_VEL
LIN {X 0,Y 446.433,Z 339.874,A -85,B 0,C 180,E1 -8605.477,E2 -8605.477} C_VEL
LIN {X 0,Y 446.42,Z 339.879,A -85,B 0,C 180,E1 -8608.7,E2 -8608.7} C_VEL
LIN {X 0,Y 446.488,Z 339.869,A -85,B 0,C 180,E1 -8611.822,E2 -8611.822} C_VEL
LIN {X 0,Y 446.462,Z 339.872,A -85,B 0,C 180,E1 -8614.848,E2 -8614.848} C_VEL
LIN {X 0,Y 446.452,Z 339.871,A -85,B 0,C 180,E1 -8618.245,E2 -8618.245} C_VEL
LIN {X 0,Y 446.461,Z 339.87,A -85,B 0,C 180,E1 -8621.649,E2 -8621.649} C_VEL
LIN {X 0,Y 446.513,Z 339.868,A -85,B 0,C 180,E1 -8624.48,E2 -8624.48} C_VEL
LIN {X 0,Y 446.523,Z 339.866,A -85,B 0,C 180,E1 -8628.193,E2 -8628.193} C_VEL
LIN {X 0,Y 446.606,Z 339.854,A -85,B 0,C 180,E1 -8631.858,E2 -8631.858} C_VEL
LIN {X 0,Y 446.65,Z 339.85,A -85,B 0,C 180,E1 -8634.583,E2 -8634.583} C_VEL
LIN {X 0,Y 446.669,Z 339.846,A -85,B 0,C 180,E1 -8638.197,E2 -8638.197} C_VEL
LIN {X 0,Y 446.799,Z 339.83,A -85,B 0,C 180,E1 -8640,E2 -8640} C_VEL
LIN {X 0,Y 446.714,Z 339.84,A -85,B 0,C 180,E1 -8642.705,E2 -8642.705} C_VEL
LIN {X 0,Y 446.641,Z 339.849,A -85,B 0,C 180,E1 -8646.324,E2 -8646.324} C_VEL
LIN {X 0,Y 446.538,Z 339.863,A -85,B 0,C 180,E1 -8649.056,E2 -8649.056} C_VEL
LIN {X 0,Y 446.527,Z 339.864,A -85,B 0,C 180,E1 -8652.73,E2 -8652.73} C_VEL
LIN {X 0,Y 446.502,Z 339.869,A -85,B 0,C 180,E1 -8656.228,E2 -8656.228} C_VEL
LIN {X 0,Y 446.475,Z 339.87,A -85,B 0,C 180,E1 -8659.303,E2 -8659.303} C_VEL
LIN {X 0,Y 446.423,Z 339.876,A -85,B 0,C 180,E1 -8662.2,E2 -8662.2} C_VEL
LIN {X 0,Y 446.463,Z 339.872,A -85,B 0,C 180,E1 -8665.152,E2 -8665.152} C_VEL
LIN {X 0,Y 446.489,Z 339.87,A -85,B 0,C 180,E1 -8668.179,E2 -8668.179} C_VEL
LIN {X 0,Y 446.424,Z 339.877,A -85,B 0,C 180,E1 -8671.775,E2 -8671.775} C_VEL
LIN {X 0,Y 446.435,Z 339.873,A -85,B 0,C 180,E1 -8674.523,E2 -8674.523} C_VEL
LIN {X 0,Y 446.435,Z 339.875,A -85,B 0,C 180,E1 -8678.082,E2 -8678.082} C_VEL
LIN {X 0,Y 446.431,Z 339.876,A -85,B 0,C 180,E1 -8680.917,E2 -8680.917} C_VEL
LIN {X 0,Y 446.406,Z 339.879,A -85,B 0,C 180,E1 -8683.846,E2 -8683.846} C_VEL
LIN {X 0,Y 446.425,Z 339.878,A -85,B 0,C 180,E1 -8686.4,E2 -8686.4} C_VEL
LIN {X 0,Y 446.477,Z 339.994,A -85,B 0,C 180,E1 -8688.155,E2 -8688.155} C_VEL
LIN {X 0,Y 448.468,Z 349.953,A -85,B 0,C 180,E1 -8691.182,E2 -8691.182} C_VEL
LIN {X 0,Y 449.735,Z 356.983,A -85,B 0,C 180,E1 -8693.229,E2 -8693.229} C_VEL
LIN {X 0,Y 449.196,Z 366.232,A -85,B 0,C 180,E1 -8695.719,E2 -8695.719} C_VEL
LIN {X 0,Y 448.387,Z 379.781,A -85,B 0,C 180,E1 -8699.266,E2 -8699.266} C_VEL
LIN {X 0,Y 447.652,Z 394.101,A -85,B 0,C 180,E1 -8702.916,E2 -8702.916} C_VEL
LIN {X 0,Y 447.049,Z 407.962,A -85,B 0,C 180,E1 -8706.366,E2 -8706.366} C_VEL
LIN {X 0,Y 446.507,Z 421.742,A -85,B 0,C 180,E1 -8709.74,E2 -8709.74} C_VEL
LIN {X 0,Y 446.188,Z 433.509,A -85,B 0,C 180,E1 -8712.586,E2 -8712.586} C_VEL
LIN {X 0,Y 446.095,Z 439.127,A -85,B 0,C 180,E1 -8713.934,E2 -8713.934} C_VEL
LIN {X 0,Y 447.497,Z 453.94,A -85,B 0,C 180,E1 -8714.399,E2 -8714.399} C_VEL
LIN {X 0,Y 448.416,Z 465.14,A -85,B 0,C 180,E1 -8714.896,E2 -8714.896} C_VEL
LIN {X 0,Y 448.484,Z 470.754,A -85,B 0,C 180,E1 -8715.189,E2 -8715.189} C_VEL
LIN {X 0,Y 447.849,Z 482.564,A -85,B 0,C 180,E1 -8715.922,E2 -8715.922} C_VEL
LIN {X 0,Y 447.266,Z 494.591,A -85,B 0,C 180,E1 -8716.884,E2 -8716.884} C_VEL
LIN {X 0,Y 446.794,Z 505.452,A -85,B 0,C 180,E1 -8717.97,E2 -8717.97} C_VEL
LIN {X 0,Y 446.35,Z 514.652,A -85,B 0,C 180,E1 -8719.109,E2 -8719.109} C_VEL
LIN {X 0,Y 445.98,Z 523.651,A -85,B 0,C 180,E1 -8720.476,E2 -8720.476} C_VEL
LIN {X 0,Y 445.86,Z 530.914,A -85,B 0,C 180,E1 -8721.844,E2 -8721.844} C_VEL
LIN {X 0,Y 445.761,Z 537.204,A -85,B 0,C 180,E1 -8723.355,E2 -8723.355} C_VEL
LIN {X 0,Y 445.793,Z 542.454,A -85,B 0,C 180,E1 -8725.026,E2 -8725.026} C_VEL
LIN {X 0,Y 445.832,Z 545.479,A -85,B 0,C 180,E1 -8726.385,E2 -8726.385} C_VEL
LIN {X 0,Y 445.818,Z 546.927,A -85,B 0,C 180,E1 -8727.289,E2 -8727.289} C_VEL
LIN {X 0,Y 445.824,Z 547.911,A -85,B 0,C 180,E1 -8728.193,E2 -8728.193} C_VEL
LIN {X 0,Y 445.998,Z 548.661,A -85,B 0,C 180,E1 -8730,E2 -8730} C_VEL
LIN {X 0,Y 446.017,Z 548.37,A -85,B 0,C 180,E1 -8730.903,E2 -8730.903} C_VEL
LIN {X 0,Y 445.872,Z 546.464,A -85,B 0,C 180,E1 -8732.71,E2 -8732.71} C_VEL
LIN {X 0,Y 445.921,Z 543.898,A -85,B 0,C 180,E1 -8734.067,E2 -8734.067} C_VEL
LIN {X 0,Y 445.85,Z 540.255,A -85,B 0,C 180,E1 -8735.427,E2 -8735.427} C_VEL
LIN {X 0,Y 445.872,Z 535.562,A -85,B 0,C 180,E1 -8736.767,E2 -8736.767} C_VEL
LIN {X 0,Y 445.902,Z 529.437,A -85,B 0,C 180,E1 -8738.155,E2 -8738.155} C_VEL
LIN {X 0,Y 446.031,Z 521.949,A -85,B 0,C 180,E1 -8739.523,E2 -8739.523} C_VEL
LIN {X 0,Y 446.341,Z 512.647,A -85,B 0,C 180,E1 -8740.892,E2 -8740.892} C_VEL
LIN {X 0,Y 446.788,Z 503.235,A -85,B 0,C 180,E1 -8742.03,E2 -8742.03} C_VEL
LIN {X 0,Y 447.132,Z 493.492,A -85,B 0,C 180,E1 -8743.011,E2 -8743.011} C_VEL
LIN {X 0,Y 447.727,Z 481.872,A -85,B 0,C 180,E1 -8743.966,E2 -8743.966} C_VEL
LIN {X 0,Y 448.345,Z 469.759,A -85,B 0,C 180,E1 -8744.757,E2 -8744.757} C_VEL
LIN {X 0,Y 448.366,Z 465.694,A -85,B 0,C 180,E1 -8744.989,E2 -8744.989} C_VEL
LIN {X 0,Y 447.663,Z 454.75,A -85,B 0,C 180,E1 -8745.544,E2 -8745.544} C_VEL
LIN {X 0,Y 446.844,Z 440.774,A -85,B 0,C 180,E1 -8746.078,E2 -8746.078} C_VEL
LIN {X 0,Y 446.04,Z 433.306,A -85,B 0,C 180,E1 -8746.321,E2 -8746.321} C_VEL
LIN {X 0,Y 446.207,Z 420.121,A -85,B 0,C 180,E1 -8749.315,E2 -8749.315} C_VEL
LIN {X 0,Y 446.437,Z 405.528,A -85,B 0,C 180,E1 -8752.687,E2 -8752.687} C_VEL
LIN {X 0,Y 446.75,Z 392.063,A -85,B 0,C 180,E1 -8755.884,E2 -8755.884} C_VEL
LIN {X 0,Y 447.12,Z 378.798,A -85,B 0,C 180,E1 -8759.161,E2 -8759.161} C_VEL
LIN {X 0,Y 447.67,Z 366.928,A -85,B 0,C 180,E1 -8762.261,E2 -8762.261} C_VEL
LIN {X 0,Y 448.691,Z 353.838,A -85,B 0,C 180,E1 -8765.971,E2 -8765.971} C_VEL
LIN {X 0,Y 448.408,Z 349.802,A -85,B 0,C 180,E1 -8767.271,E2 -8767.271} C_VEL
LIN {X 0,Y 447.16,Z 343.328,A -85,B 0,C 180,E1 -8769.634,E2 -8769.634} C_VEL
LIN {X 0,Y 446.436,Z 339.878,A -85,B 0,C 180,E1 -8771.117,E2 -8771.117} C_VEL
LIN {X 0,Y 446.405,Z 339.882,A -85,B 0,C 180,E1 -8773.846,E2 -8773.846} C_VEL
LIN {X 0,Y 446.403,Z 339.88,A -85,B 0,C 180,E1 -8776.403,E2 -8776.403} C_VEL
LIN {X 0,Y 446.43,Z 339.876,A -85,B 0,C 180,E1 -8779.082,E2 -8779.082} C_VEL
LIN {X 0,Y 446.431,Z 339.875,A -85,B 0,C 180,E1 -8782.123,E2 -8782.123} C_VEL
LIN {X 0,Y 446.434,Z 339.876,A -85,B 0,C 180,E1 -8785.477,E2 -8785.477} C_VEL
LIN {X 0,Y 446.42,Z 339.877,A -85,B 0,C 180,E1 -8788.7,E2 -8788.7} C_VEL
LIN {X 0,Y 446.489,Z 339.867,A -85,B 0,C 180,E1 -8791.821,E2 -8791.821} C_VEL
LIN {X 0,Y 446.448,Z 339.874,A -85,B 0,C 180,E1 -8794.847,E2 -8794.847} C_VEL
LIN {X 0,Y 446.452,Z 339.875,A -85,B 0,C 180,E1 -8798.245,E2 -8798.245} C_VEL
LIN {X 0,Y 446.461,Z 339.875,A -85,B 0,C 180,E1 -8801.649,E2 -8801.649} C_VEL
LIN {X 0,Y 446.487,Z 339.871,A -85,B 0,C 180,E1 -8803.511,E2 -8803.511} C_VEL
LIN {X 0,Y 450.051,Z 351.255,A -85,B 0,C 180,E1 -8804.337,E2 -8804.337} C_VEL
LIN {X 0,Y 450.175,Z 355.254,A -85,B 0,C 180,E1 -8804.609,E2 -8804.609} C_VEL
LIN {X 0,Y 449.732,Z 365.715,A -85,B 0,C 180,E1 -8805.405,E2 -8805.405} C_VEL
LIN {X 0,Y 449.115,Z 376.523,A -85,B 0,C 180,E1 -8806.424,E2 -8806.424} C_VEL
LIN {X 0,Y 448.616,Z 386.181,A -85,B 0,C 180,E1 -8807.56,E2 -8807.56} C_VEL
LIN {X 0,Y 448.113,Z 394.078,A -85,B 0,C 180,E1 -8808.694,E2 -8808.694} C_VEL
LIN {X 0,Y 447.643,Z 401.776,A -85,B 0,C 180,E1 -8810.055,E2 -8810.055} C_VEL
LIN {X 0,Y 447.215,Z 407.934,A -85,B 0,C 180,E1 -8811.414,E2 -8811.414} C_VEL
LIN {X 0,Y 446.91,Z 412.766,A -85,B 0,C 180,E1 -8812.773,E2 -8812.773} C_VEL
LIN {X 0,Y 446.634,Z 416.466,A -85,B 0,C 180,E1 -8814.129,E2 -8814.129} C_VEL
LIN {X 0,Y 446.389,Z 419.139,A -85,B 0,C 180,E1 -8815.485,E2 -8815.485} C_VEL
LIN {X 0,Y 446.298,Z 420.359,A -85,B 0,C 180,E1 -8816.388,E2 -8816.388} C_VEL
LIN {X 0,Y 446.197,Z 421.62,A -85,B 0,C 180,E1 -8818.195,E2 -8818.195} C_VEL
LIN {X 0,Y 446.184,Z 421.651,A -85,B 0,C 180,E1 -8819.097,E2 -8819.097} C_VEL
LIN {X 0,Y 446.116,Z 420.491,A -85,B 0,C 180,E1 -8820.903,E2 -8820.903} C_VEL
LIN {X 0,Y 446.196,Z 419.318,A -85,B 0,C 180,E1 -8821.805,E2 -8821.805} C_VEL
LIN {X 0,Y 446.258,Z 416.755,A -85,B 0,C 180,E1 -8823.16,E2 -8823.16} C_VEL
LIN {X 0,Y 446.389,Z 413.195,A -85,B 0,C 180,E1 -8824.515,E2 -8824.515} C_VEL
LIN {X 0,Y 446.618,Z 408.541,A -85,B 0,C 180,E1 -8825.871,E2 -8825.871} C_VEL
LIN {X 0,Y 447.058,Z 401.535,A -85,B 0,C 180,E1 -8827.446,E2 -8827.446} C_VEL
LIN {X 0,Y 447.4,Z 393.924,A -85,B 0,C 180,E1 -8828.81,E2 -8828.81} C_VEL
LIN {X 0,Y 447.754,Z 386.211,A -85,B 0,C 180,E1 -8829.942,E2 -8829.942} C_VEL
LIN {X 0,Y 448.23,Z 376.854,A -85,B 0,C 180,E1 -8831.074,E2 -8831.074} C_VEL
LIN {X 0,Y 448.743,Z 365.225,A -85,B 0,C 180,E1 -8832.206,E2 -8832.206} C_VEL
LIN {X 0,Y 449.05,Z 356.76,A -85,B 0,C 180,E1 -8832.88,E2 -8832.88} C_VEL
LIN {X 0,Y 449.269,Z 350.307,A -85,B 0,C 180,E1 -8833.324,E2 -8833.324} C_VEL
LIN {X 0,Y 446.513,Z 339.868,A -85,B 0,C 180,E1 -8834.033,E2 -8834.033} C_VEL
LIN {X 0,Y 446.492,Z 339.866,A -85,B 0,C 180,E1 -8836.459,E2 -8836.459} C_VEL
LIN {X 0,Y 446.472,Z 339.872,A -85,B 0,C 180,E1 -8839.303,E2 -8839.303} C_VEL
LIN {X 0,Y 446.422,Z 339.876,A -85,B 0,C 180,E1 -8842.199,E2 -8842.199} C_VEL
LIN {X 0,Y 446.461,Z 339.872,A -85,B 0,C 180,E1 -8845.152,E2 -8845.152} C_VEL
LIN {X 0,Y 446.487,Z 339.869,A -85,B 0,C 180,E1 -8848.178,E2 -8848.178} C_VEL
LIN {X 0,Y 446.423,Z 339.876,A -85,B 0,C 180,E1 -8851.775,E2 -8851.775} C_VEL
LIN {X 0,Y 446.432,Z 339.874,A -85,B 0,C 180,E1 -8854.523,E2 -8854.523} C_VEL
LIN {X 0,Y 446.439,Z 339.873,A -85,B 0,C 180,E1 -8858.083,E2 -8858.083} C_VEL
LIN {X 0,Y 446.445,Z 339.874,A -85,B 0,C 180,E1 -8860.92,E2 -8860.92} C_VEL
LIN {X 0,Y 446.404,Z 339.879,A -85,B 0,C 180,E1 -8863.846,E2 -8863.846} C_VEL
LIN {X 0,Y 446.426,Z 339.876,A -85,B 0,C 180,E1 -8866.4,E2 -8866.4} C_VEL
LIN {X 0,Y 446.449,Z 339.873,A -85,B 0,C 180,E1 -8869.802,E2 -8869.802} C_VEL
LIN {X 0,Y 446.411,Z 339.876,A -85,B 0,C 180,E1 -8872.121,E2 -8872.121} C_VEL
LIN {X 0,Y 446.43,Z 339.873,A -85,B 0,C 180,E1 -8875.477,E2 -8875.477} C_VEL
LIN {X 0,Y 446.417,Z 339.877,A -85,B 0,C 180,E1 -8878.7,E2 -8878.7} C_VEL
LIN {X 0,Y 446.486,Z 339.87,A -85,B 0,C 180,E1 -8881.821,E2 -8881.821} C_VEL
LIN {X 0,Y 446.46,Z 339.875,A -85,B 0,C 180,E1 -8884.848,E2 -8884.848} C_VEL
LIN {X 0,Y 446.449,Z 339.874,A -85,B 0,C 180,E1 -8888.245,E2 -8888.245} C_VEL
LIN {X 0,Y 446.459,Z 339.87,A -85,B 0,C 180,E1 -8891.649,E2 -8891.649} C_VEL
LIN {X 0,Y 446.509,Z 339.866,A -85,B 0,C 180,E1 -8894.48,E2 -8894.48} C_VEL
LIN {X 0,Y 446.519,Z 339.865,A -85,B 0,C 180,E1 -8898.193,E2 -8898.193} C_VEL
LIN {X 0,Y 446.601,Z 339.854,A -85,B 0,C 180,E1 -8901.858,E2 -8901.858} C_VEL
LIN {X 0,Y 446.639,Z 339.85,A -85,B 0,C 180,E1 -8904.489,E2 -8904.489} C_VEL
LIN {X 0,Y 446.011,Z 339.934,A -85,B 0,C 180,E1 -8905.241,E2 -8905.241} C_VEL
LIN {X 0,Y 443.185,Z 340.289,A -85,B 0,C 180,E1 -8906.464,E2 -8906.464} C_VEL
LIN {X 0,Y 440.764,Z 340.588,A -85,B 0,C 180,E1 -8907.45,E2 -8907.45} C_VEL
LIN {X 0,Y 439.709,Z 340.715,A -85,B 0,C 180,E1 -8908.213,E2 -8908.213} C_VEL
LIN {X 0,Y 439.616,Z 340.723,A -85,B 0,C 180,E1 -8908.471,E2 -8908.471} C_VEL
LIN {X 0,Y 439.764,Z 340.709,A -85,B 0,C 180,E1 -8910,E2 -8910} C_VEL
LIN {X 0,Y 439.658,Z 340.718,A -85,B 0,C 180,E1 -8912.749,E2 -8912.749} C_VEL
LIN {X 0,Y 439.613,Z 340.726,A -85,B 0,C 180,E1 -8916.425,E2 -8916.425} C_VEL
LIN {X 0,Y 439.502,Z 340.74,A -85,B 0,C 180,E1 -8919.202,E2 -8919.202} C_VEL
LIN {X 0,Y 439.467,Z 340.742,A -85,B 0,C 180,E1 -8922.938,E2 -8922.938} C_VEL
LIN {X 0,Y 439.449,Z 340.743,A -85,B 0,C 180,E1 -8926.349,E2 -8926.349} C_VEL
LIN {X 0,Y 439.404,Z 340.753,A -85,B 0,C 180,E1 -8929.626,E2 -8929.626} C_VEL
LIN {X 0,Y 439.366,Z 340.755,A -85,B 0,C 180,E1 -8932.576,E2 -8932.576} C_VEL
LIN {X 0,Y 439.407,Z 340.751,A -85,B 0,C 180,E1 -8935.585,E2 -8935.585} C_VEL
LIN {X 0,Y 439.419,Z 340.749,A -85,B 0,C 180,E1 -8938.674,E2 -8938.674} C_VEL
LIN {X 0,Y 439.372,Z 340.754,A -85,B 0,C 180,E1 -8942.031,E2 -8942.031} C_VEL
LIN {X 0,Y 439.396,Z 340.755,A -85,B 0,C 180,E1 -8945.341,E2 -8945.341} C_VEL
LIN {X 0,Y 439.385,Z 340.753,A -85,B 0,C 180,E1 -8948.595,E2 -8948.595} C_VEL
LIN {X 0,Y 439.397,Z 340.752,A -85,B 0,C 180,E1 -8951.258,E2 -8951.258} C_VEL
LIN {X 0,Y 439.412,Z 340.751,A -85,B 0,C 180,E1 -8954.728,E2 -8954.728} C_VEL
LIN {X 0,Y 439.399,Z 340.752,A -85,B 0,C 180,E1 -8957.796,E2 -8957.796} C_VEL
LIN {X 0,Y 439.428,Z 340.746,A -85,B 0,C 180,E1 -8960.228,E2 -8960.228} C_VEL
LIN {X 0,Y 439.377,Z 340.752,A -85,B 0,C 180,E1 -8963.713,E2 -8963.713} C_VEL
LIN {X 0,Y 439.376,Z 340.755,A -85,B 0,C 180,E1 -8967.054,E2 -8967.054} C_VEL
LIN {X 0,Y 439.386,Z 340.754,A -85,B 0,C 180,E1 -8970.275,E2 -8970.275} C_VEL
LIN {X 0,Y 439.434,Z 340.749,A -85,B 0,C 180,E1 -8973.397,E2 -8973.397} C_VEL
LIN {X 0,Y 439.391,Z 340.751,A -85,B 0,C 180,E1 -8976.43,E2 -8976.43} C_VEL
LIN {X 0,Y 439.393,Z 340.75,A -85,B 0,C 180,E1 -8979.397,E2 -8979.397} C_VEL
LIN {X 0,Y 439.435,Z 340.747,A -85,B 0,C 180,E1 -8982.31,E2 -8982.31} C_VEL
LIN {X 0,Y 439.453,Z 340.744,A -85,B 0,C 180,E1 -8985.174,E2 -8985.174} C_VEL
LIN {X 0,Y 439.489,Z 340.741,A -85,B 0,C 180,E1 -8988.002,E2 -8988.002} C_VEL
LIN {X 0,Y 439.553,Z 340.732,A -85,B 0,C 180,E1 -8991.727,E2 -8991.727} C_VEL
LIN {X 0,Y 439.626,Z 340.724,A -85,B 0,C 180,E1 -8994.496,E2 -8994.496} C_VEL
LIN {X 0,Y 439.639,Z 340.722,A -85,B 0,C 180,E1 -8998.168,E2 -8998.168} C_VEL
LIN {X 0,Y 439.768,Z 340.706,A -85,B 0,C 180,E1 -9000,E2 -9000} C_VEL
LIN {X 0,Y 439.661,Z 340.719,A -85,B 0,C 180,E1 -9002.749,E2 -9002.749} C_VEL
LIN {X 0,Y 439.611,Z 340.725,A -85,B 0,C 180,E1 -9006.425,E2 -9006.425} C_VEL
LIN {X 0,Y 439.501,Z 340.739,A -85,B 0,C 180,E1 -9009.202,E2 -9009.202} C_VEL
LIN {X 0,Y 439.471,Z 340.741,A -85,B 0,C 180,E1 -9012.938,E2 -9012.938} C_VEL
LIN {X 0,Y 439.453,Z 340.746,A -85,B 0,C 180,E1 -9016.349,E2 -9016.349} C_VEL
LIN {X 0,Y 439.408,Z 340.751,A -85,B 0,C 180,E1 -9019.626,E2 -9019.626} C_VEL
LIN {X 0,Y 439.37,Z 340.756,A -85,B 0,C 180,E1 -9022.575,E2 -9022.575} C_VEL
LIN {X 0,Y 439.41,Z 340.75,A -85,B 0,C 180,E1 -9025.585,E2 -9025.585} C_VEL
LIN {X 0,Y 439.422,Z 340.748,A -85,B 0,C 180,E1 -9028.673,E2 -9028.673} C_VEL
LIN {X 0,Y 439.375,Z 340.758,A -85,B 0,C 180,E1 -9032.03,E2 -9032.03} C_VEL
LIN {X 0,Y 439.401,Z 340.751,A -85,B 0,C 180,E1 -9035.341,E2 -9035.341} C_VEL
LIN {X 0,Y 439.393,Z 340.753,A -85,B 0,C 180,E1 -9038.594,E2 -9038.594} C_VEL
LIN {X 0,Y 439.392,Z 340.754,A -85,B 0,C 180,E1 -9041.257,E2 -9041.257} C_VEL
LIN {X 0,Y 439.406,Z 340.753,A -85,B 0,C 180,E1 -9044.729,E2 -9044.729} C_VEL
LIN {X 0,Y 439.437,Z 340.895,A -85,B 0,C 180,E1 -9047.874,E2 -9047.874} C_VEL
LIN {X 0,Y 441.617,Z 351.818,A -85,B 0,C 180,E1 -9051.242,E2 -9051.242} C_VEL
LIN {X 0,Y 442.805,Z 358.402,A -85,B 0,C 180,E1 -9053.19,E2 -9053.19} C_VEL
LIN {X 0,Y 442.174,Z 367.755,A -85,B 0,C 180,E1 -9055.741,E2 -9055.741} C_VEL
LIN {X 0,Y 441.454,Z 379.38,A -85,B 0,C 180,E1 -9058.842,E2 -9058.842} C_VEL
LIN {X 0,Y 440.764,Z 391.288,A -85,B 0,C 180,E1 -9061.941,E2 -9061.941} C_VEL
LIN {X 0,Y 440.119,Z 405.375,A -85,B 0,C 180,E1 -9065.534,E2 -9065.534} C_VEL
LIN {X 0,Y 439.564,Z 418.866,A -85,B 0,C 180,E1 -9068.915,E2 -9068.915} C_VEL
LIN {X 0,Y 439.22,Z 430.621,A -85,B 0,C 180,E1 -9071.819,E2 -9071.819} C_VEL
LIN {X 0,Y 439.019,Z 438.256,A -85,B 0,C 180,E1 -9073.691,E2 -9073.691} C_VEL
LIN {X 0,Y 440.493,Z 454.062,A -85,B 0,C 180,E1 -9074.215,E2 -9074.215} C_VEL
LIN {X 0,Y 441.426,Z 465.946,A -85,B 0,C 180,E1 -9074.77,E2 -9074.77} C_VEL
LIN {X 0,Y 441.428,Z 472.281,A -85,B 0,C 180,E1 -9075.124,E2 -9075.124} C_VEL
LIN {X 0,Y 440.745,Z 484.291,A -85,B 0,C 180,E1 -9075.926,E2 -9075.926} C_VEL
LIN {X 0,Y 440.162,Z 495.785,A -85,B 0,C 180,E1 -9076.902,E2 -9076.902} C_VEL
LIN {X 0,Y 439.652,Z 506.174,A -85,B 0,C 180,E1 -9078.006,E2 -9078.006} C_VEL
LIN {X 0,Y 439.249,Z 515.103,A -85,B 0,C 180,E1 -9079.164,E2 -9079.164} C_VEL
LIN {X 0,Y 438.889,Z 523.843,A -85,B 0,C 180,E1 -9080.553,E2 -9080.553} C_VEL
LIN {X 0,Y 438.772,Z 530.837,A -85,B 0,C 180,E1 -9081.943,E2 -9081.943} C_VEL
LIN {X 0,Y 438.692,Z 537.237,A -85,B 0,C 180,E1 -9083.561,E2 -9083.561} C_VEL
LIN {X 0,Y 438.744,Z 541.398,A -85,B 0,C 180,E1 -9084.945,E2 -9084.945} C_VEL
LIN {X 0,Y 438.79,Z 544.442,A -85,B 0,C 180,E1 -9086.327,E2 -9086.327} C_VEL
LIN {X 0,Y 438.777,Z 545.904,A -85,B 0,C 180,E1 -9087.246,E2 -9087.246} C_VEL
LIN {X 0,Y 438.789,Z 546.894,A -85,B 0,C 180,E1 -9088.164,E2 -9088.164} C_VEL
LIN {X 0,Y 438.976,Z 547.646,A -85,B 0,C 180,E1 -9090,E2 -9090} C_VEL
LIN {X 0,Y 438.995,Z 547.361,A -85,B 0,C 180,E1 -9090.917,E2 -9090.917} C_VEL
LIN {X 0,Y 438.831,Z 545.44,A -85,B 0,C 180,E1 -9092.754,E2 -9092.754} C_VEL
LIN {X 0,Y 438.878,Z 542.868,A -85,B 0,C 180,E1 -9094.132,E2 -9094.132} C_VEL
LIN {X 0,Y 438.782,Z 539.217,A -85,B 0,C 180,E1 -9095.515,E2 -9095.515} C_VEL
LIN {X 0,Y 438.782,Z 534.356,A -85,B 0,C 180,E1 -9096.918,E2 -9096.918} C_VEL
LIN {X 0,Y 438.859,Z 528.379,A -85,B 0,C 180,E1 -9098.287,E2 -9098.287} C_VEL
LIN {X 0,Y 438.963,Z 520.894,A -85,B 0,C 180,E1 -9099.678,E2 -9099.678} C_VEL
LIN {X 0,Y 439.302,Z 511.615,A -85,B 0,C 180,E1 -9101.068,E2 -9101.068} C_VEL
LIN {X 0,Y 439.788,Z 502.319,A -85,B 0,C 180,E1 -9102.213,E2 -9102.213} C_VEL
LIN {X 0,Y 440.101,Z 493.486,A -85,B 0,C 180,E1 -9103.13,E2 -9103.13} C_VEL
LIN {X 0,Y 440.702,Z 482.522,A -85,B 0,C 180,E1 -9104.075,E2 -9104.075} C_VEL
LIN {X 0,Y 441.353,Z 470.991,A -85,B 0,C 180,E1 -9104.879,E2 -9104.879} C_VEL
LIN {X 0,Y 441.278,Z 465.08,A -85,B 0,C 180,E1 -9105.236,E2 -9105.236} C_VEL
LIN {X 0,Y 440.688,Z 452.686,A -85,B 0,C 180,E1 -9105.873,E2 -9105.873} C_VEL
LIN {X 0,Y 439.863,Z 439.719,A -85,B 0,C 180,E1 -9106.385,E2 -9106.385} C_VEL
LIN {X 0,Y 438.95,Z 431.876,A -85,B 0,C 180,E1 -9106.668,E2 -9106.668} C_VEL
LIN {X 0,Y 439.149,Z 419.068,A -85,B 0,C 180,E1 -9109.638,E2 -9109.638} C_VEL
LIN {X 0,Y 439.411,Z 404.54,A -85,B 0,C 180,E1 -9113.07,E2 -9113.07} C_VEL
LIN {X 0,Y 439.713,Z 392.343,A -85,B 0,C 180,E1 -9116.035,E2 -9116.035} C_VEL
LIN {X 0,Y 440.101,Z 380.038,A -85,B 0,C 180,E1 -9119.147,E2 -9119.147} C_VEL
LIN {X 0,Y 440.687,Z 368.227,A -85,B 0,C 180,E1 -9122.303,E2 -9122.303} C_VEL
LIN {X 0,Y 441.788,Z 355.288,A -85,B 0,C 180,E1 -9126.058,E2 -9126.058} C_VEL
LIN {X 0,Y 441.555,Z 351.624,A -85,B 0,C 180,E1 -9127.266,E2 -9127.266} C_VEL
LIN {X 0,Y 440.169,Z 344.432,A -85,B 0,C 180,E1 -9129.968,E2 -9129.968} C_VEL
LIN {X 0,Y 439.391,Z 340.755,A -85,B 0,C 180,E1 -9131.563,E2 -9131.563} C_VEL
LIN {X 0,Y 439.405,Z 340.752,A -85,B 0,C 180,E1 -9135.271,E2 -9135.271} C_VEL
LIN {X 0,Y 439.392,Z 340.755,A -85,B 0,C 180,E1 -9138.743,E2 -9138.743} C_VEL
LIN {X 0,Y 439.386,Z 340.755,A -85,B 0,C 180,E1 -9141.606,E2 -9141.606} C_VEL
LIN {X 0,Y 439.405,Z 340.752,A -85,B 0,C 180,E1 -9144.844,E2 -9144.844} C_VEL
LIN {X 0,Y 439.377,Z 340.756,A -85,B 0,C 180,E1 -9148.14,E2 -9148.14} C_VEL
LIN {X 0,Y 439.436,Z 340.747,A -85,B 0,C 180,E1 -9151.598,E2 -9151.598} C_VEL
LIN {X 0,Y 439.402,Z 340.753,A -85,B 0,C 180,E1 -9154.415,E2 -9154.415} C_VEL
LIN {X 0,Y 439.368,Z 340.758,A -85,B 0,C 180,E1 -9157.425,E2 -9157.425} C_VEL
LIN {X 0,Y 439.446,Z 340.749,A -85,B 0,C 180,E1 -9160.663,E2 -9160.663} C_VEL
LIN {X 0,Y 439.422,Z 340.766,A -85,B 0,C 180,E1 -9163.179,E2 -9163.179} C_VEL
LIN {X 0,Y 443.245,Z 352.608,A -85,B 0,C 180,E1 -9164.07,E2 -9164.07} C_VEL
LIN {X 0,Y 443.53,Z 355.828,A -85,B 0,C 180,E1 -9164.3,E2 -9164.3} C_VEL
LIN {X 0,Y 442.995,Z 367.222,A -85,B 0,C 180,E1 -9165.178,E2 -9165.178} C_VEL
LIN {X 0,Y 442.354,Z 377.96,A -85,B 0,C 180,E1 -9166.213,E2 -9166.213} C_VEL
LIN {X 0,Y 441.826,Z 387.519,A -85,B 0,C 180,E1 -9167.366,E2 -9167.366} C_VEL
LIN {X 0,Y 441.289,Z 395.337,A -85,B 0,C 180,E1 -9168.517,E2 -9168.517} C_VEL
LIN {X 0,Y 440.749,Z 402.972,A -85,B 0,C 180,E1 -9169.898,E2 -9169.898} C_VEL
LIN {X 0,Y 440.319,Z 409.108,A -85,B 0,C 180,E1 -9171.278,E2 -9171.278} C_VEL
LIN {X 0,Y 439.979,Z 413.924,A -85,B 0,C 180,E1 -9172.658,E2 -9172.658} C_VEL
LIN {X 0,Y 439.674,Z 417.605,A -85,B 0,C 180,E1 -9174.036,E2 -9174.036} C_VEL
LIN {X 0,Y 439.398,Z 420.26,A -85,B 0,C 180,E1 -9175.413,E2 -9175.413} C_VEL
LIN {X 0,Y 439.24,Z 422.272,A -85,B 0,C 180,E1 -9177.249,E2 -9177.249} C_VEL
LIN {X 0,Y 439.206,Z 422.689,A -85,B 0,C 180,E1 -9178.166,E2 -9178.166} C_VEL
LIN {X 0,Y 439.18,Z 422.694,A -85,B 0,C 180,E1 -9179.083,E2 -9179.083} C_VEL
LIN {X 0,Y 439.093,Z 421.499,A -85,B 0,C 180,E1 -9180.917,E2 -9180.917} C_VEL
LIN {X 0,Y 439.175,Z 420.303,A -85,B 0,C 180,E1 -9181.834,E2 -9181.834} C_VEL
LIN {X 0,Y 439.246,Z 417.707,A -85,B 0,C 180,E1 -9183.21,E2 -9183.21} C_VEL
LIN {X 0,Y 439.372,Z 414.114,A -85,B 0,C 180,E1 -9184.587,E2 -9184.587} C_VEL
LIN {X 0,Y 439.627,Z 409.421,A -85,B 0,C 180,E1 -9185.964,E2 -9185.964} C_VEL
LIN {X 0,Y 440.081,Z 402.395,A -85,B 0,C 180,E1 -9187.558,E2 -9187.558} C_VEL
LIN {X 0,Y 440.441,Z 394.713,A -85,B 0,C 180,E1 -9188.95,E2 -9188.95} C_VEL
LIN {X 0,Y 440.812,Z 386.958,A -85,B 0,C 180,E1 -9190.1,E2 -9190.1} C_VEL
LIN {X 0,Y 441.307,Z 377.539,A -85,B 0,C 180,E1 -9191.25,E2 -9191.25} C_VEL
LIN {X 0,Y 441.846,Z 365.858,A -85,B 0,C 180,E1 -9192.4,E2 -9192.4} C_VEL
LIN {X 0,Y 442.073,Z 358.498,A -85,B 0,C 180,E1 -9193,E2 -9193} C_VEL
LIN {X 0,Y 442.168,Z 350.872,A -85,B 0,C 180,E1 -9193.542,E2 -9193.542} C_VEL
LIN {X 0,Y 439.432,Z 340.749,A -85,B 0,C 180,E1 -9194.235,E2 -9194.235} C_VEL
LIN {X 0,Y 439.452,Z 340.743,A -85,B 0,C 180,E1 -9196.73,E2 -9196.73} C_VEL
LIN {X 0,Y 439.405,Z 340.749,A -85,B 0,C 180,E1 -9199.626,E2 -9199.626} C_VEL
LIN {X 0,Y 439.368,Z 340.756,A -85,B 0,C 180,E1 -9202.575,E2 -9202.575} C_VEL
LIN {X 0,Y 439.408,Z 340.751,A -85,B 0,C 180,E1 -9205.585,E2 -9205.585} C_VEL
LIN {X 0,Y 439.421,Z 340.749,A -85,B 0,C 180,E1 -9208.673,E2 -9208.673} C_VEL
LIN {X 0,Y 439.374,Z 340.754,A -85,B 0,C 180,E1 -9212.03,E2 -9212.03} C_VEL
LIN {X 0,Y 439.397,Z 340.751,A -85,B 0,C 180,E1 -9215.34,E2 -9215.34} C_VEL
LIN {X 0,Y 439.4,Z 340.754,A -85,B 0,C 180,E1 -9218.593,E2 -9218.593} C_VEL
LIN {X 0,Y 439.401,Z 340.751,A -85,B 0,C 180,E1 -9221.258,E2 -9221.258} C_VEL
LIN {X 0,Y 439.405,Z 340.751,A -85,B 0,C 180,E1 -9224.729,E2 -9224.729} C_VEL
LIN {X 0,Y 439.4,Z 340.751,A -85,B 0,C 180,E1 -9227.796,E2 -9227.796} C_VEL
LIN {X 0,Y 439.431,Z 340.746,A -85,B 0,C 180,E1 -9230.228,E2 -9230.228} C_VEL
LIN {X 0,Y 439.375,Z 340.751,A -85,B 0,C 180,E1 -9233.713,E2 -9233.713} C_VEL
LIN {X 0,Y 439.373,Z 340.754,A -85,B 0,C 180,E1 -9237.054,E2 -9237.054} C_VEL
LIN {X 0,Y 439.384,Z 340.755,A -85,B 0,C 180,E1 -9240.274,E2 -9240.274} C_VEL
LIN {X 0,Y 439.431,Z 340.748,A -85,B 0,C 180,E1 -9243.396,E2 -9243.396} C_VEL
LIN {X 0,Y 439.388,Z 340.754,A -85,B 0,C 180,E1 -9246.43,E2 -9246.43} C_VEL
LIN {X 0,Y 439.39,Z 340.751,A -85,B 0,C 180,E1 -9249.397,E2 -9249.397} C_VEL
LIN {X 0,Y 439.433,Z 340.75,A -85,B 0,C 180,E1 -9252.31,E2 -9252.31} C_VEL
LIN {X 0,Y 439.449,Z 340.744,A -85,B 0,C 180,E1 -9255.174,E2 -9255.174} C_VEL
LIN {X 0,Y 439.485,Z 340.742,A -85,B 0,C 180,E1 -9258.001,E2 -9258.001} C_VEL
LIN {X 0,Y 439.549,Z 340.733,A -85,B 0,C 180,E1 -9261.726,E2 -9261.726} C_VEL
LIN {X 0,Y 439.619,Z 340.726,A -85,B 0,C 180,E1 -9264.496,E2 -9264.496} C_VEL
LIN {X 0,Y 439.637,Z 340.724,A -85,B 0,C 180,E1 -9268.168,E2 -9268.168} C_VEL
LIN {X 0,Y 439.616,Z 340.723,A -85,B 0,C 180,E1 -9268.471,E2 -9268.471} C_VEL
LIN {X 0,Y 438.931,Z 340.808,A -85,B 0,C 180,E1 -9269.235,E2 -9269.235} C_VEL
LIN {X 0,Y 436.076,Z 341.164,A -85,B 0,C 180,E1 -9270.478,E2 -9270.478} C_VEL
LIN {X 0,Y 433.682,Z 341.464,A -85,B 0,C 180,E1 -9271.481,E2 -9271.481} C_VEL
LIN {X 0,Y 432.67,Z 341.59,A -85,B 0,C 180,E1 -9272.256,E2 -9272.256} C_VEL
LIN {X 0,Y 432.595,Z 341.598,A -85,B 0,C 180,E1 -9272.518,E2 -9272.518} C_VEL
LIN {X 0,Y 432.595,Z 341.601,A -85,B 0,C 180,E1 -9275.594,E2 -9275.594} C_VEL
LIN {X 0,Y 432.493,Z 341.613,A -85,B 0,C 180,E1 -9278.41,E2 -9278.41} C_VEL
LIN {X 0,Y 432.461,Z 341.617,A -85,B 0,C 180,E1 -9282.197,E2 -9282.197} C_VEL
LIN {X 0,Y 432.432,Z 341.62,A -85,B 0,C 180,E1 -9286.039,E2 -9286.039} C_VEL
LIN {X 0,Y 432.388,Z 341.628,A -85,B 0,C 180,E1 -9289.486,E2 -9289.486} C_VEL
LIN {X 0,Y 432.321,Z 341.634,A -85,B 0,C 180,E1 -9292.964,E2 -9292.964} C_VEL
LIN {X 0,Y 432.366,Z 341.63,A -85,B 0,C 180,E1 -9296.033,E2 -9296.033} C_VEL
LIN {X 0,Y 432.345,Z 341.63,A -85,B 0,C 180,E1 -9299.188,E2 -9299.188} C_VEL
LIN {X 0,Y 432.325,Z 341.63,A -85,B 0,C 180,E1 -9302.443,E2 -9302.443} C_VEL
LIN {X 0,Y 432.346,Z 341.63,A -85,B 0,C 180,E1 -9305.632,E2 -9305.632} C_VEL
LIN {X 0,Y 432.352,Z 341.63,A -85,B 0,C 180,E1 -9309.343,E2 -9309.343} C_VEL
LIN {X 0,Y 432.373,Z 341.628,A -85,B 0,C 180,E1 -9311.793,E2 -9311.793} C_VEL
LIN {X 0,Y 432.381,Z 341.626,A -85,B 0,C 180,E1 -9314.342,E2 -9314.342} C_VEL
LIN {X 0,Y 432.336,Z 341.63,A -85,B 0,C 180,E1 -9318.203,E2 -9318.203} C_VEL
LIN {X 0,Y 432.345,Z 341.632,A -85,B 0,C 180,E1 -9321.286,E2 -9321.286} C_VEL
LIN {X 0,Y 432.347,Z 341.629,A -85,B 0,C 180,E1 -9324.368,E2 -9324.368} C_VEL
LIN {X 0,Y 432.326,Z 341.632,A -85,B 0,C 180,E1 -9327.557,E2 -9327.557} C_VEL
LIN {X 0,Y 432.347,Z 341.63,A -85,B 0,C 180,E1 -9330.813,E2 -9330.813} C_VEL
LIN {X 0,Y 432.368,Z 341.627,A -85,B 0,C 180,E1 -9333.968,E2 -9333.968} C_VEL
LIN {X 0,Y 432.323,Z 341.636,A -85,B 0,C 180,E1 -9337.036,E2 -9337.036} C_VEL
LIN {X 0,Y 432.391,Z 341.625,A -85,B 0,C 180,E1 -9340.515,E2 -9340.515} C_VEL
LIN {X 0,Y 432.435,Z 341.618,A -85,B 0,C 180,E1 -9343.961,E2 -9343.961} C_VEL
LIN {X 0,Y 432.464,Z 341.615,A -85,B 0,C 180,E1 -9347.804,E2 -9347.804} C_VEL
LIN {X 0,Y 432.497,Z 341.611,A -85,B 0,C 180,E1 -9351.591,E2 -9351.591} C_VEL
LIN {X 0,Y 432.602,Z 341.598,A -85,B 0,C 180,E1 -9354.406,E2 -9354.406} C_VEL
LIN {X 0,Y 432.609,Z 341.597,A -85,B 0,C 180,E1 -9358.138,E2 -9358.138} C_VEL
LIN {X 0,Y 432.738,Z 341.581,A -85,B 0,C 180,E1 -9360,E2 -9360} C_VEL
LIN {X 0,Y 432.61,Z 341.597,A -85,B 0,C 180,E1 -9362.794,E2 -9362.794} C_VEL
LIN {X 0,Y 432.561,Z 341.604,A -85,B 0,C 180,E1 -9366.531,E2 -9366.531} C_VEL
LIN {X 0,Y 432.445,Z 341.617,A -85,B 0,C 180,E1 -9369.353,E2 -9369.353} C_VEL
LIN {X 0,Y 432.436,Z 341.618,A -85,B 0,C 180,E1 -9372.804,E2 -9372.804} C_VEL
LIN {X 0,Y 432.418,Z 341.621,A -85,B 0,C 180,E1 -9376.479,E2 -9376.479} C_VEL
LIN {X 0,Y 432.345,Z 341.632,A -85,B 0,C 180,E1 -9379.96,E2 -9379.96} C_VEL
LIN {X 0,Y 432.324,Z 341.633,A -85,B 0,C 180,E1 -9382.964,E2 -9382.964} C_VEL
LIN {X 0,Y 432.369,Z 341.628,A -85,B 0,C 180,E1 -9386.032,E2 -9386.032} C_VEL
LIN {X 0,Y 432.348,Z 341.629,A -85,B 0,C 180,E1 -9389.187,E2 -9389.187} C_VEL
LIN {X 0,Y 432.328,Z 341.631,A -85,B 0,C 180,E1 -9392.443,E2 -9392.443} C_VEL
LIN {X 0,Y 432.35,Z 341.632,A -85,B 0,C 180,E1 -9395.632,E2 -9395.632} C_VEL
LIN {X 0,Y 432.355,Z 341.629,A -85,B 0,C 180,E1 -9398.716,E2 -9398.716} C_VEL
LIN {X 0,Y 432.337,Z 341.631,A -85,B 0,C 180,E1 -9401.797,E2 -9401.797} C_VEL
LIN {X 0,Y 432.337,Z 341.634,A -85,B 0,C 180,E1 -9404.347,E2 -9404.347} C_VEL
LIN {X 0,Y 432.367,Z 341.653,A -85,B 0,C 180,E1 -9407.54,E2 -9407.54} C_VEL
LIN {X 0,Y 434.521,Z 352.417,A -85,B 0,C 180,E1 -9410.929,E2 -9410.929} C_VEL
LIN {X 0,Y 435.732,Z 358.728,A -85,B 0,C 180,E1 -9412.836,E2 -9412.836} C_VEL
LIN {X 0,Y 435.654,Z 363.242,A -85,B 0,C 180,E1 -9414.115,E2 -9414.115} C_VEL
LIN {X 0,Y 434.732,Z 375.494,A -85,B 0,C 180,E1 -9417.47,E2 -9417.47} C_VEL
LIN {X 0,Y 433.959,Z 388.453,A -85,B 0,C 180,E1 -9420.931,E2 -9420.931} C_VEL
LIN {X 0,Y 433.277,Z 400.285,A -85,B 0,C 180,E1 -9424.026,E2 -9424.026} C_VEL
LIN {X 0,Y 432.749,Z 412.076,A -85,B 0,C 180,E1 -9427.06,E2 -9427.06} C_VEL
LIN {X 0,Y 432.249,Z 425.903,A -85,B 0,C 180,E1 -9430.568,E2 -9430.568} C_VEL
LIN {X 0,Y 431.938,Z 437.514,A -85,B 0,C 180,E1 -9433.472,E2 -9433.472} C_VEL
LIN {X 0,Y 433.272,Z 451.723,A -85,B 0,C 180,E1 -9433.937,E2 -9433.937} C_VEL
LIN {X 0,Y 434.284,Z 465.314,A -85,B 0,C 180,E1 -9434.573,E2 -9434.573} C_VEL
LIN {X 0,Y 434.501,Z 470.691,A -85,B 0,C 180,E1 -9434.881,E2 -9434.881} C_VEL
LIN {X 0,Y 433.788,Z 482.809,A -85,B 0,C 180,E1 -9435.695,E2 -9435.695} C_VEL
LIN {X 0,Y 433.188,Z 493.841,A -85,B 0,C 180,E1 -9436.633,E2 -9436.633} C_VEL
LIN {X 0,Y 432.854,Z 502.968,A -85,B 0,C 180,E1 -9437.584,E2 -9437.584} C_VEL
LIN {X 0,Y 432.291,Z 512.226,A -85,B 0,C 180,E1 -9438.75,E2 -9438.75} C_VEL
LIN {X 0,Y 431.841,Z 521.299,A -85,B 0,C 180,E1 -9440.161,E2 -9440.161} C_VEL
LIN {X 0,Y 431.715,Z 528.646,A -85,B 0,C 180,E1 -9441.575,E2 -9441.575} C_VEL
LIN {X 0,Y 431.639,Z 534.665,A -85,B 0,C 180,E1 -9443.033,E2 -9443.033} C_VEL
LIN {X 0,Y 431.63,Z 539.068,A -85,B 0,C 180,E1 -9444.393,E2 -9444.393} C_VEL
LIN {X 0,Y 431.715,Z 541.462,A -85,B 0,C 180,E1 -9445.331,E2 -9445.331} C_VEL
LIN {X 0,Y 431.75,Z 543.392,A -85,B 0,C 180,E1 -9446.267,E2 -9446.267} C_VEL
LIN {X 0,Y 431.738,Z 544.869,A -85,B 0,C 180,E1 -9447.201,E2 -9447.201} C_VEL
LIN {X 0,Y 431.755,Z 545.866,A -85,B 0,C 180,E1 -9448.134,E2 -9448.134} C_VEL
LIN {X 0,Y 431.8,Z 546.447,A -85,B 0,C 180,E1 -9449.067,E2 -9449.067} C_VEL
LIN {X 0,Y 431.953,Z 546.625,A -85,B 0,C 180,E1 -9450,E2 -9450} C_VEL
LIN {X 0,Y 431.971,Z 546.349,A -85,B 0,C 180,E1 -9450.932,E2 -9450.932} C_VEL
LIN {X 0,Y 431.789,Z 544.421,A -85,B 0,C 180,E1 -9452.799,E2 -9452.799} C_VEL
LIN {X 0,Y 431.836,Z 541.844,A -85,B 0,C 180,E1 -9454.2,E2 -9454.2} C_VEL
LIN {X 0,Y 431.716,Z 538.186,A -85,B 0,C 180,E1 -9455.605,E2 -9455.605} C_VEL
LIN {X 0,Y 431.705,Z 532.588,A -85,B 0,C 180,E1 -9457.225,E2 -9457.225} C_VEL
LIN {X 0,Y 431.798,Z 526.231,A -85,B 0,C 180,E1 -9458.659,E2 -9458.659} C_VEL
LIN {X 0,Y 431.915,Z 518.438,A -85,B 0,C 180,E1 -9460.074,E2 -9460.074} C_VEL
LIN {X 0,Y 432.328,Z 508.897,A -85,B 0,C 180,E1 -9461.487,E2 -9461.487} C_VEL
LIN {X 0,Y 432.751,Z 499.967,A -85,B 0,C 180,E1 -9462.577,E2 -9462.577} C_VEL
LIN {X 0,Y 433.359,Z 489.931,A -85,B 0,C 180,E1 -9463.601,E2 -9463.601} C_VEL
LIN {X 0,Y 433.958,Z 478.724,A -85,B 0,C 180,E1 -9464.538,E2 -9464.538} C_VEL
LIN {X 0,Y 434.542,Z 468.501,A -85,B 0,C 180,E1 -9465.237,E2 -9465.237} C_VEL
LIN {X 0,Y 433.936,Z 456.853,A -85,B 0,C 180,E1 -9465.921,E2 -9465.921} C_VEL
LIN {X 0,Y 433.311,Z 442.989,A -85,B 0,C 180,E1 -9466.55,E2 -9466.55} C_VEL
LIN {X 0,Y 431.931,Z 430.532,A -85,B 0,C 180,E1 -9467.008,E2 -9467.008} C_VEL
LIN {X 0,Y 432.148,Z 415.963,A -85,B 0,C 180,E1 -9470.466,E2 -9470.466} C_VEL
LIN {X 0,Y 432.468,Z 400.477,A -85,B 0,C 180,E1 -9474.233,E2 -9474.233} C_VEL
LIN {X 0,Y 432.851,Z 387.278,A -85,B 0,C 180,E1 -9477.564,E2 -9477.564} C_VEL
LIN {X 0,Y 433.326,Z 375.354,A -85,B 0,C 180,E1 -9480.729,E2 -9480.729} C_VEL
LIN {X 0,Y 433.902,Z 365.816,A -85,B 0,C 180,E1 -9483.416,E2 -9483.416} C_VEL
LIN {X 0,Y 434.854,Z 356.925,A -85,B 0,C 180,E1 -9486.09,E2 -9486.09} C_VEL
LIN {X 0,Y 434.731,Z 353.77,A -85,B 0,C 180,E1 -9487.147,E2 -9487.147} C_VEL
LIN {X 0,Y 433.472,Z 346.913,A -85,B 0,C 180,E1 -9489.749,E2 -9489.749} C_VEL
LIN {X 0,Y 432.372,Z 341.629,A -85,B 0,C 180,E1 -9492.106,E2 -9492.106} C_VEL
LIN {X 0,Y 432.336,Z 341.633,A -85,B 0,C 180,E1 -9495.665,E2 -9495.665} C_VEL
LIN {X 0,Y 432.336,Z 341.633,A -85,B 0,C 180,E1 -9498.398,E2 -9498.398} C_VEL
LIN {X 0,Y 432.349,Z 341.63,A -85,B 0,C 180,E1 -9501.851,E2 -9501.851} C_VEL
LIN {X 0,Y 432.345,Z 341.631,A -85,B 0,C 180,E1 -9505.323,E2 -9505.323} C_VEL
LIN {X 0,Y 432.325,Z 341.632,A -85,B 0,C 180,E1 -9508.654,E2 -9508.654} C_VEL
LIN {X 0,Y 432.385,Z 341.624,A -85,B 0,C 180,E1 -9511.877,E2 -9511.877} C_VEL
LIN {X 0,Y 432.35,Z 341.63,A -85,B 0,C 180,E1 -9514.998,E2 -9514.998} C_VEL
LIN {X 0,Y 432.362,Z 341.631,A -85,B 0,C 180,E1 -9518.046,E2 -9518.046} C_VEL
LIN {X 0,Y 432.391,Z 341.627,A -85,B 0,C 180,E1 -9521.03,E2 -9521.03} C_VEL
LIN {X 0,Y 432.415,Z 341.639,A -85,B 0,C 180,E1 -9522.822,E2 -9522.822} C_VEL
LIN {X 0,Y 436.361,Z 353.57,A -85,B 0,C 180,E1 -9523.746,E2 -9523.746} C_VEL
LIN {X 0,Y 436.903,Z 356.823,A -85,B 0,C 180,E1 -9524.001,E2 -9524.001} C_VEL
LIN {X 0,Y 436.353,Z 367.454,A -85,B 0,C 180,E1 -9524.827,E2 -9524.827} C_VEL
LIN {X 0,Y 435.602,Z 379.396,A -85,B 0,C 180,E1 -9525.995,E2 -9525.995} C_VEL
LIN {X 0,Y 435.033,Z 388.895,A -85,B 0,C 180,E1 -9527.166,E2 -9527.166} C_VEL
LIN {X 0,Y 434.462,Z 396.678,A -85,B 0,C 180,E1 -9528.334,E2 -9528.334} C_VEL
LIN {X 0,Y 433.88,Z 404.279,A -85,B 0,C 180,E1 -9529.736,E2 -9529.736} C_VEL
LIN {X 0,Y 433.426,Z 410.345,A -85,B 0,C 180,E1 -9531.139,E2 -9531.139} C_VEL
LIN {X 0,Y 433.046,Z 415.106,A -85,B 0,C 180,E1 -9532.54,E2 -9532.54} C_VEL
LIN {X 0,Y 432.729,Z 418.742,A -85,B 0,C 180,E1 -9533.94,E2 -9533.94} C_VEL
LIN {X 0,Y 432.407,Z 421.381,A -85,B 0,C 180,E1 -9535.338,E2 -9535.338} C_VEL
LIN {X 0,Y 432.295,Z 422.569,A -85,B 0,C 180,E1 -9536.271,E2 -9536.271} C_VEL
LIN {X 0,Y 432.212,Z 423.757,A -85,B 0,C 180,E1 -9538.136,E2 -9538.136} C_VEL
LIN {X 0,Y 432.174,Z 423.739,A -85,B 0,C 180,E1 -9539.068,E2 -9539.068} C_VEL
LIN {X 0,Y 432.138,Z 423.313,A -85,B 0,C 180,E1 -9540,E2 -9540} C_VEL
LIN {X 0,Y 432.07,Z 422.503,A -85,B 0,C 180,E1 -9540.932,E2 -9540.932} C_VEL
LIN {X 0,Y 432.154,Z 421.281,A -85,B 0,C 180,E1 -9541.864,E2 -9541.864} C_VEL
LIN {X 0,Y 432.232,Z 418.645,A -85,B 0,C 180,E1 -9543.262,E2 -9543.262} C_VEL
LIN {X 0,Y 432.352,Z 415.008,A -85,B 0,C 180,E1 -9544.662,E2 -9544.662} C_VEL
LIN {X 0,Y 432.634,Z 410.258,A -85,B 0,C 180,E1 -9546.061,E2 -9546.061} C_VEL
LIN {X 0,Y 433.104,Z 403.216,A -85,B 0,C 180,E1 -9547.671,E2 -9547.671} C_VEL
LIN {X 0,Y 433.461,Z 395.42,A -85,B 0,C 180,E1 -9549.096,E2 -9549.096} C_VEL
LIN {X 0,Y 433.876,Z 387.594,A -85,B 0,C 180,E1 -9550.264,E2 -9550.264} C_VEL
LIN {X 0,Y 434.363,Z 378.079,A -85,B 0,C 180,E1 -9551.432,E2 -9551.432} C_VEL
LIN {X 0,Y 434.921,Z 366.315,A -85,B 0,C 180,E1 -9552.6,E2 -9552.6} C_VEL
LIN {X 0,Y 435.291,Z 357.325,A -85,B 0,C 180,E1 -9553.324,E2 -9553.324} C_VEL
LIN {X 0,Y 435.361,Z 352.81,A -85,B 0,C 180,E1 -9553.644,E2 -9553.644} C_VEL
LIN {X 0,Y 432.396,Z 341.624,A -85,B 0,C 180,E1 -9554.441,E2 -9554.441} C_VEL
LIN {X 0,Y 432.393,Z 341.625,A -85,B 0,C 180,E1 -9557.012,E2 -9557.012} C_VEL
LIN {X 0,Y 432.342,Z 341.628,A -85,B 0,C 180,E1 -9559.96,E2 -9559.96} C_VEL
LIN {X 0,Y 432.322,Z 341.635,A -85,B 0,C 180,E1 -9562.964,E2 -9562.964} C_VEL
LIN {X 0,Y 432.368,Z 341.627,A -85,B 0,C 180,E1 -9566.032,E2 -9566.032} C_VEL
LIN {X 0,Y 432.346,Z 341.631,A -85,B 0,C 180,E1 -9569.187,E2 -9569.187} C_VEL
LIN {X 0,Y 432.326,Z 341.632,A -85,B 0,C 180,E1 -9572.443,E2 -9572.443} C_VEL
LIN {X 0,Y 432.347,Z 341.627,A -85,B 0,C 180,E1 -9575.632,E2 -9575.632} C_VEL
LIN {X 0,Y 432.362,Z 341.631,A -85,B 0,C 180,E1 -9578.717,E2 -9578.717} C_VEL
LIN {X 0,Y 432.368,Z 341.627,A -85,B 0,C 180,E1 -9581.793,E2 -9581.793} C_VEL
LIN {X 0,Y 432.335,Z 341.633,A -85,B 0,C 180,E1 -9584.347,E2 -9584.347} C_VEL
LIN {X 0,Y 432.327,Z 341.634,A -85,B 0,C 180,E1 -9587.015,E2 -9587.015} C_VEL
LIN {X 0,Y 432.338,Z 341.63,A -85,B 0,C 180,E1 -9589.82,E2 -9589.82} C_VEL
LIN {X 0,Y 432.308,Z 341.634,A -85,B 0,C 180,E1 -9593.022,E2 -9593.022} C_VEL
LIN {X 0,Y 432.36,Z 341.628,A -85,B 0,C 180,E1 -9595.996,E2 -9595.996} C_VEL
LIN {X 0,Y 432.349,Z 341.629,A -85,B 0,C 180,E1 -9599.489,E2 -9599.489} C_VEL
LIN {X 0,Y 432.394,Z 341.626,A -85,B 0,C 180,E1 -9602.928,E2 -9602.928} C_VEL
LIN {X 0,Y 432.373,Z 341.626,A -85,B 0,C 180,E1 -9606.023,E2 -9606.023} C_VEL
LIN {X 0,Y 432.352,Z 341.628,A -85,B 0,C 180,E1 -9609.046,E2 -9609.046} C_VEL
LIN {X 0,Y 432.379,Z 341.626,A -85,B 0,C 180,E1 -9612.011,E2 -9612.011} C_VEL
LIN {X 0,Y 432.397,Z 341.623,A -85,B 0,C 180,E1 -9614.926,E2 -9614.926} C_VEL
LIN {X 0,Y 432.46,Z 341.618,A -85,B 0,C 180,E1 -9617.803,E2 -9617.803} C_VEL
LIN {X 0,Y 432.493,Z 341.613,A -85,B 0,C 180,E1 -9621.59,E2 -9621.59} C_VEL
LIN {X 0,Y 432.596,Z 341.602,A -85,B 0,C 180,E1 -9624.406,E2 -9624.406} C_VEL
LIN {X 0,Y 432.607,Z 341.6,A -85,B 0,C 180,E1 -9628.138,E2 -9628.138} C_VEL
LIN {X 0,Y 432.733,Z 341.585,A -85,B 0,C 180,E1 -9630,E2 -9630} C_VEL
LIN {X 0,Y 432.595,Z 341.598,A -85,B 0,C 180,E1 -9632.518,E2 -9632.518} C_VEL
LIN {X 0,Y 431.94,Z 341.682,A -85,B 0,C 180,E1 -9633.294,E2 -9633.294} C_VEL
LIN {X 0,Y 429.063,Z 342.039,A -85,B 0,C 180,E1 -9634.554,E2 -9634.554} C_VEL
LIN {X 0,Y 426.629,Z 342.345,A -85,B 0,C 180,E1 -9635.571,E2 -9635.571} C_VEL
LIN {X 0,Y 425.599,Z 342.471,A -85,B 0,C 180,E1 -9636.358,E2 -9636.358} C_VEL
LIN {X 0,Y 425.524,Z 342.48,A -85,B 0,C 180,E1 -9636.624,E2 -9636.624} C_VEL
LIN {X 0,Y 425.403,Z 342.495,A -85,B 0,C 180,E1 -9639.509,E2 -9639.509} C_VEL
LIN {X 0,Y 425.394,Z 342.495,A -85,B 0,C 180,E1 -9642.904,E2 -9642.904} C_VEL
LIN {X 0,Y 425.363,Z 342.497,A -85,B 0,C 180,E1 -9646.605,E2 -9646.605} C_VEL
LIN {X 0,Y 425.33,Z 342.506,A -85,B 0,C 180,E1 -9649.636,E2 -9649.636} C_VEL
LIN {X 0,Y 425.308,Z 342.508,A -85,B 0,C 180,E1 -9653.365,E2 -9653.365} C_VEL
LIN {X 0,Y 425.349,Z 342.502,A -85,B 0,C 180,E1 -9656.844,E2 -9656.844} C_VEL
LIN {X 0,Y 425.293,Z 342.512,A -85,B 0,C 180,E1 -9659.72,E2 -9659.72} C_VEL
LIN {X 0,Y 425.284,Z 342.509,A -85,B 0,C 180,E1 -9663.048,E2 -9663.048} C_VEL
LIN {X 0,Y 425.284,Z 342.508,A -85,B 0,C 180,E1 -9665.929,E2 -9665.929} C_VEL
LIN {X 0,Y 425.3,Z 342.51,A -85,B 0,C 180,E1 -9669.044,E2 -9669.044} C_VEL
LIN {X 0,Y 425.333,Z 342.504,A -85,B 0,C 180,E1 -9672.646,E2 -9672.646} C_VEL
LIN {X 0,Y 425.297,Z 342.509,A -85,B 0,C 180,E1 -9675.282,E2 -9675.282} C_VEL
LIN {X 0,Y 425.277,Z 342.51,A -85,B 0,C 180,E1 -9678.622,E2 -9678.622} C_VEL
LIN {X 0,Y 425.309,Z 342.509,A -85,B 0,C 180,E1 -9681.103,E2 -9681.103} C_VEL
LIN {X 0,Y 425.303,Z 342.508,A -85,B 0,C 180,E1 -9684.665,E2 -9684.665} C_VEL
LIN {X 0,Y 425.268,Z 342.511,A -85,B 0,C 180,E1 -9688.073,E2 -9688.073} C_VEL
LIN {X 0,Y 425.335,Z 342.505,A -85,B 0,C 180,E1 -9691.368,E2 -9691.368} C_VEL
LIN {X 0,Y 425.299,Z 342.508,A -85,B 0,C 180,E1 -9694.555,E2 -9694.555} C_VEL
LIN {X 0,Y 425.292,Z 342.507,A -85,B 0,C 180,E1 -9697.662,E2 -9697.662} C_VEL
LIN {X 0,Y 425.366,Z 342.502,A -85,B 0,C 180,E1 -9700.704,E2 -9700.704} C_VEL
LIN {X 0,Y 425.393,Z 342.495,A -85,B 0,C 180,E1 -9703.689,E2 -9703.689} C_VEL
LIN {X 0,Y 425.417,Z 342.493,A -85,B 0,C 180,E1 -9707.598,E2 -9707.598} C_VEL
LIN {X 0,Y 425.448,Z 342.489,A -85,B 0,C 180,E1 -9711.45,E2 -9711.45} C_VEL
LIN {X 0,Y 425.559,Z 342.475,A -85,B 0,C 180,E1 -9714.313,E2 -9714.313} C_VEL
LIN {X 0,Y 425.578,Z 342.473,A -85,B 0,C 180,E1 -9718.107,E2 -9718.107} C_VEL
LIN {X 0,Y 425.707,Z 342.457,A -85,B 0,C 180,E1 -9720,E2 -9720} C_VEL
LIN {X 0,Y 425.561,Z 342.475,A -85,B 0,C 180,E1 -9722.84,E2 -9722.84} C_VEL
LIN {X 0,Y 425.553,Z 342.477,A -85,B 0,C 180,E1 -9725.687,E2 -9725.687} C_VEL
LIN {X 0,Y 425.413,Z 342.495,A -85,B 0,C 180,E1 -9728.551,E2 -9728.551} C_VEL
LIN {X 0,Y 425.417,Z 342.496,A -85,B 0,C 180,E1 -9732.402,E2 -9732.402} C_VEL
LIN {X 0,Y 425.394,Z 342.498,A -85,B 0,C 180,E1 -9736.312,E2 -9736.312} C_VEL
LIN {X 0,Y 425.334,Z 342.504,A -85,B 0,C 180,E1 -9739.636,E2 -9739.636} C_VEL
LIN {X 0,Y 425.312,Z 342.506,A -85,B 0,C 180,E1 -9743.365,E2 -9743.365} C_VEL
LIN {X 0,Y 425.352,Z 342.501,A -85,B 0,C 180,E1 -9746.844,E2 -9746.844} C_VEL
LIN {X 0,Y 425.296,Z 342.508,A -85,B 0,C 180,E1 -9749.719,E2 -9749.719} C_VEL
LIN {X 0,Y 425.287,Z 342.506,A -85,B 0,C 180,E1 -9753.048,E2 -9753.048} C_VEL
LIN {X 0,Y 425.289,Z 342.51,A -85,B 0,C 180,E1 -9755.929,E2 -9755.929} C_VEL
LIN {X 0,Y 425.305,Z 342.507,A -85,B 0,C 180,E1 -9759.044,E2 -9759.044} C_VEL
LIN {X 0,Y 425.279,Z 342.513,A -85,B 0,C 180,E1 -9762.653,E2 -9762.653} C_VEL
LIN {X 0,Y 425.273,Z 342.513,A -85,B 0,C 180,E1 -9766.045,E2 -9766.045} C_VEL
LIN {X 0,Y 425.349,Z 342.667,A -85,B 0,C 180,E1 -9767.293,E2 -9767.293} C_VEL
LIN {X 0,Y 427.4,Z 353.018,A -85,B 0,C 180,E1 -9770.611,E2 -9770.611} C_VEL
LIN {X 0,Y 428.696,Z 359.662,A -85,B 0,C 180,E1 -9772.657,E2 -9772.657} C_VEL
LIN {X 0,Y 428.764,Z 363.722,A -85,B 0,C 180,E1 -9773.836,E2 -9773.836} C_VEL
LIN {X 0,Y 427.808,Z 375.659,A -85,B 0,C 180,E1 -9777.171,E2 -9777.171} C_VEL
LIN {X 0,Y 427.006,Z 387.55,A -85,B 0,C 180,E1 -9780.411,E2 -9780.411} C_VEL
LIN {X 0,Y 426.316,Z 399.369,A -85,B 0,C 180,E1 -9783.57,E2 -9783.57} C_VEL
LIN {X 0,Y 425.768,Z 411.132,A -85,B 0,C 180,E1 -9786.661,E2 -9786.661} C_VEL
LIN {X 0,Y 425.201,Z 425.642,A -85,B 0,C 180,E1 -9790.414,E2 -9790.414} C_VEL
LIN {X 0,Y 424.843,Z 436.662,A -85,B 0,C 180,E1 -9793.235,E2 -9793.235} C_VEL
LIN {X 0,Y 426.288,Z 451.892,A -85,B 0,C 180,E1 -9793.754,E2 -9793.754} C_VEL
LIN {X 0,Y 427.162,Z 464.613,A -85,B 0,C 180,E1 -9794.37,E2 -9794.37} C_VEL
LIN {X 0,Y 427.591,Z 469.033,A -85,B 0,C 180,E1 -9794.631,E2 -9794.631} C_VEL
LIN {X 0,Y 426.917,Z 481.295,A -85,B 0,C 180,E1 -9795.46,E2 -9795.46} C_VEL
LIN {X 0,Y 426.244,Z 492.404,A -85,B 0,C 180,E1 -9796.411,E2 -9796.411} C_VEL
LIN {X 0,Y 425.834,Z 501.905,A -85,B 0,C 180,E1 -9797.41,E2 -9797.41} C_VEL
LIN {X 0,Y 425.261,Z 510.957,A -85,B 0,C 180,E1 -9798.561,E2 -9798.561} C_VEL
LIN {X 0,Y 424.798,Z 520.081,A -85,B 0,C 180,E1 -9799.996,E2 -9799.996} C_VEL
LIN {X 0,Y 424.632,Z 527.466,A -85,B 0,C 180,E1 -9801.433,E2 -9801.433} C_VEL
LIN {X 0,Y 424.582,Z 533.543,A -85,B 0,C 180,E1 -9802.916,E2 -9802.916} C_VEL
LIN {X 0,Y 424.575,Z 537.975,A -85,B 0,C 180,E1 -9804.3,E2 -9804.3} C_VEL
LIN {X 0,Y 424.671,Z 540.386,A -85,B 0,C 180,E1 -9805.253,E2 -9805.253} C_VEL
LIN {X 0,Y 424.711,Z 542.327,A -85,B 0,C 180,E1 -9806.205,E2 -9806.205} C_VEL
LIN {X 0,Y 424.7,Z 543.819,A -85,B 0,C 180,E1 -9807.154,E2 -9807.154} C_VEL
LIN {X 0,Y 424.721,Z 544.831,A -85,B 0,C 180,E1 -9808.103,E2 -9808.103} C_VEL
LIN {X 0,Y 424.794,Z 545.418,A -85,B 0,C 180,E1 -9809.052,E2 -9809.052} C_VEL
LIN {X 0,Y 424.931,Z 545.598,A -85,B 0,C 180,E1 -9810,E2 -9810} C_VEL
LIN {X 0,Y 424.947,Z 545.333,A -85,B 0,C 180,E1 -9810.948,E2 -9810.948} C_VEL
LIN {X 0,Y 424.753,Z 544.568,A -85,B 0,C 180,E1 -9811.896,E2 -9811.896} C_VEL
LIN {X 0,Y 424.747,Z 543.406,A -85,B 0,C 180,E1 -9812.845,E2 -9812.845} C_VEL
LIN {X 0,Y 424.794,Z 540.833,A -85,B 0,C 180,E1 -9814.27,E2 -9814.27} C_VEL
LIN {X 0,Y 424.652,Z 537.169,A -85,B 0,C 180,E1 -9815.699,E2 -9815.699} C_VEL
LIN {X 0,Y 424.634,Z 532.386,A -85,B 0,C 180,E1 -9817.13,E2 -9817.13} C_VEL
LIN {X 0,Y 424.708,Z 526.349,A -85,B 0,C 180,E1 -9818.565,E2 -9818.565} C_VEL
LIN {X 0,Y 424.82,Z 518.874,A -85,B 0,C 180,E1 -9820.003,E2 -9820.003} C_VEL
LIN {X 0,Y 425.239,Z 509.69,A -85,B 0,C 180,E1 -9821.439,E2 -9821.439} C_VEL
LIN {X 0,Y 425.708,Z 499.536,A -85,B 0,C 180,E1 -9822.735,E2 -9822.735} C_VEL
LIN {X 0,Y 426.362,Z 489.134,A -85,B 0,C 180,E1 -9823.828,E2 -9823.828} C_VEL
LIN {X 0,Y 427.054,Z 478.103,A -85,B 0,C 180,E1 -9824.779,E2 -9824.779} C_VEL
LIN {X 0,Y 427.532,Z 468.076,A -85,B 0,C 180,E1 -9825.493,E2 -9825.493} C_VEL
LIN {X 0,Y 427.068,Z 456.773,A -85,B 0,C 180,E1 -9826.185,E2 -9826.185} C_VEL
LIN {X 0,Y 426.432,Z 442.465,A -85,B 0,C 180,E1 -9826.866,E2 -9826.866} C_VEL
LIN {X 0,Y 424.835,Z 429.131,A -85,B 0,C 180,E1 -9827.386,E2 -9827.386} C_VEL
LIN {X 0,Y 425.071,Z 414.97,A -85,B 0,C 180,E1 -9830.823,E2 -9830.823} C_VEL
LIN {X 0,Y 425.413,Z 400.62,A -85,B 0,C 180,E1 -9834.394,E2 -9834.394} C_VEL
LIN {X 0,Y 425.859,Z 387.506,A -85,B 0,C 180,E1 -9837.789,E2 -9837.789} C_VEL
LIN {X 0,Y 426.481,Z 374.454,A -85,B 0,C 180,E1 -9841.358,E2 -9841.358} C_VEL
LIN {X 0,Y 427.298,Z 363.195,A -85,B 0,C 180,E1 -9844.676,E2 -9844.676} C_VEL
LIN {X 0,Y 427.971,Z 357.663,A -85,B 0,C 180,E1 -9846.422,E2 -9846.422} C_VEL
LIN {X 0,Y 427.365,Z 352.644,A -85,B 0,C 180,E1 -9848.234,E2 -9848.234} C_VEL
LIN {X 0,Y 426.194,Z 346.749,A -85,B 0,C 180,E1 -9850.663,E2 -9850.663} C_VEL
LIN {X 0,Y 425.293,Z 342.512,A -85,B 0,C 180,E1 -9852.722,E2 -9852.722} C_VEL
LIN {X 0,Y 425.265,Z 342.515,A -85,B 0,C 180,E1 -9856.044,E2 -9856.044} C_VEL
LIN {X 0,Y 425.278,Z 342.514,A -85,B 0,C 180,E1 -9858.621,E2 -9858.621} C_VEL
LIN {X 0,Y 425.313,Z 342.507,A -85,B 0,C 180,E1 -9861.103,E2 -9861.103} C_VEL
LIN {X 0,Y 425.304,Z 342.509,A -85,B 0,C 180,E1 -9864.664,E2 -9864.664} C_VEL
LIN {X 0,Y 425.269,Z 342.513,A -85,B 0,C 180,E1 -9868.073,E2 -9868.073} C_VEL
LIN {X 0,Y 425.335,Z 342.505,A -85,B 0,C 180,E1 -9871.368,E2 -9871.368} C_VEL
LIN {X 0,Y 425.357,Z 342.5,A -85,B 0,C 180,E1 -9873.505,E2 -9873.505} C_VEL
LIN {X 0,Y 425.309,Z 342.507,A -85,B 0,C 180,E1 -9876.635,E2 -9876.635} C_VEL
LIN {X 0,Y 425.333,Z 342.507,A -85,B 0,C 180,E1 -9880.364,E2 -9880.364} C_VEL
LIN {X 0,Y 425.376,Z 342.561,A -85,B 0,C 180,E1 -9882.435,E2 -9882.435} C_VEL
LIN {X 0,Y 429.778,Z 355.668,A -85,B 0,C 180,E1 -9883.501,E2 -9883.501} C_VEL
LIN {X 0,Y 430.233,Z 357.229,A -85,B 0,C 180,E1 -9883.639,E2 -9883.639} C_VEL
LIN {X 0,Y 429.77,Z 367.869,A -85,B 0,C 180,E1 -9884.468,E2 -9884.468} C_VEL
LIN {X 0,Y 429.095,Z 378.834,A -85,B 0,C 180,E1 -9885.539,E2 -9885.539} C_VEL
LIN {X 0,Y 428.417,Z 388.611,A -85,B 0,C 180,E1 -9886.723,E2 -9886.723} C_VEL
LIN {X 0,Y 427.743,Z 396.626,A -85,B 0,C 180,E1 -9887.907,E2 -9887.907} C_VEL
LIN {X 0,Y 427.107,Z 404.43,A -85,B 0,C 180,E1 -9889.332,E2 -9889.332} C_VEL
LIN {X 0,Y 426.692,Z 409.741,A -85,B 0,C 180,E1 -9890.52,E2 -9890.52} C_VEL
LIN {X 0,Y 426.212,Z 415.062,A -85,B 0,C 180,E1 -9892.002,E2 -9892.002} C_VEL
LIN {X 0,Y 425.891,Z 418.838,A -85,B 0,C 180,E1 -9893.367,E2 -9893.367} C_VEL
LIN {X 0,Y 425.582,Z 420.917,A -85,B 0,C 180,E1 -9894.313,E2 -9894.313} C_VEL
LIN {X 0,Y 425.422,Z 422.534,A -85,B 0,C 180,E1 -9895.262,E2 -9895.262} C_VEL
LIN {X 0,Y 425.238,Z 424.456,A -85,B 0,C 180,E1 -9897.158,E2 -9897.158} C_VEL
LIN {X 0,Y 425.215,Z 424.83,A -85,B 0,C 180,E1 -9898.106,E2 -9898.106} C_VEL
LIN {X 0,Y 425.167,Z 424.783,A -85,B 0,C 180,E1 -9899.053,E2 -9899.053} C_VEL
LIN {X 0,Y 425.129,Z 424.332,A -85,B 0,C 180,E1 -9900,E2 -9900} C_VEL
LIN {X 0,Y 425.046,Z 423.505,A -85,B 0,C 180,E1 -9900.947,E2 -9900.947} C_VEL
LIN {X 0,Y 425.132,Z 422.257,A -85,B 0,C 180,E1 -9901.895,E2 -9901.895} C_VEL
LIN {X 0,Y 425.216,Z 419.58,A -85,B 0,C 180,E1 -9903.316,E2 -9903.316} C_VEL
LIN {X 0,Y 425.333,Z 415.898,A -85,B 0,C 180,E1 -9904.739,E2 -9904.739} C_VEL
LIN {X 0,Y 425.641,Z 411.09,A -85,B 0,C 180,E1 -9906.161,E2 -9906.161} C_VEL
LIN {X 0,Y 426.126,Z 404.011,A -85,B 0,C 180,E1 -9907.791,E2 -9907.791} C_VEL
LIN {X 0,Y 426.499,Z 396.122,A -85,B 0,C 180,E1 -9909.245,E2 -9909.245} C_VEL
LIN {X 0,Y 426.946,Z 388.218,A -85,B 0,C 180,E1 -9910.432,E2 -9910.432} C_VEL
LIN {X 0,Y 427.464,Z 377.547,A -85,B 0,C 180,E1 -9911.739,E2 -9911.739} C_VEL
LIN {X 0,Y 428.013,Z 366.759,A -85,B 0,C 180,E1 -9912.807,E2 -9912.807} C_VEL
LIN {X 0,Y 428.442,Z 356.901,A -85,B 0,C 180,E1 -9913.6,E2 -9913.6} C_VEL
LIN {X 0,Y 428.488,Z 354.746,A -85,B 0,C 180,E1 -9913.751,E2 -9913.751} C_VEL
LIN {X 0,Y 425.371,Z 342.499,A -85,B 0,C 180,E1 -9914.655,E2 -9914.655} C_VEL
LIN {X 0,Y 425.337,Z 342.506,A -85,B 0,C 180,E1 -9917.303,E2 -9917.303} C_VEL
LIN {X 0,Y 425.298,Z 342.506,A -85,B 0,C 180,E1 -9920.305,E2 -9920.305} C_VEL
LIN {X 0,Y 425.31,Z 342.506,A -85,B 0,C 180,E1 -9923.365,E2 -9923.365} C_VEL
LIN {X 0,Y 425.351,Z 342.502,A -85,B 0,C 180,E1 -9926.844,E2 -9926.844} C_VEL
LIN {X 0,Y 425.294,Z 342.509,A -85,B 0,C 180,E1 -9929.719,E2 -9929.719} C_VEL
LIN {X 0,Y 425.285,Z 342.512,A -85,B 0,C 180,E1 -9933.048,E2 -9933.048} C_VEL
LIN {X 0,Y 425.286,Z 342.506,A -85,B 0,C 180,E1 -9935.929,E2 -9935.929} C_VEL
LIN {X 0,Y 425.315,Z 342.506,A -85,B 0,C 180,E1 -9939.046,E2 -9939.046} C_VEL
LIN {X 0,Y 425.317,Z 342.505,A -85,B 0,C 180,E1 -9941.962,E2 -9941.962} C_VEL
LIN {X 0,Y 425.292,Z 342.51,A -85,B 0,C 180,E1 -9945.282,E2 -9945.282} C_VEL
LIN {X 0,Y 425.278,Z 342.511,A -85,B 0,C 180,E1 -9948.621,E2 -9948.621} C_VEL
LIN {X 0,Y 425.311,Z 342.506,A -85,B 0,C 180,E1 -9951.102,E2 -9951.102} C_VEL
LIN {X 0,Y 425.3,Z 342.51,A -85,B 0,C 180,E1 -9954.664,E2 -9954.664} C_VEL
LIN {X 0,Y 425.266,Z 342.513,A -85,B 0,C 180,E1 -9958.073,E2 -9958.073} C_VEL
LIN {X 0,Y 425.332,Z 342.503,A -85,B 0,C 180,E1 -9961.368,E2 -9961.368} C_VEL
LIN {X 0,Y 425.297,Z 342.509,A -85,B 0,C 180,E1 -9964.555,E2 -9964.555} C_VEL
LIN {X 0,Y 425.289,Z 342.508,A -85,B 0,C 180,E1 -9967.661,E2 -9967.661} C_VEL
LIN {X 0,Y 425.366,Z 342.499,A -85,B 0,C 180,E1 -9970.704,E2 -9970.704} C_VEL
LIN {X 0,Y 425.39,Z 342.496,A -85,B 0,C 180,E1 -9973.688,E2 -9973.688} C_VEL
LIN {X 0,Y 425.413,Z 342.494,A -85,B 0,C 180,E1 -9977.598,E2 -9977.598} C_VEL
LIN {X 0,Y 425.444,Z 342.49,A -85,B 0,C 180,E1 -9981.45,E2 -9981.45} C_VEL
LIN {X 0,Y 425.552,Z 342.479,A -85,B 0,C 180,E1 -9984.313,E2 -9984.313} C_VEL
LIN {X 0,Y 425.576,Z 342.476,A -85,B 0,C 180,E1 -9988.107,E2 -9988.107} C_VEL
LIN {X 0,Y 425.703,Z 342.46,A -85,B 0,C 180,E1 -9990,E2 -9990} C_VEL
LIN {X 0,Y 425.559,Z 342.474,A -85,B 0,C 180,E1 -9992.84,E2 -9992.84} C_VEL
LIN {X 0,Y 425.524,Z 342.48,A -85,B 0,C 180,E1 -9996.624,E2 -9996.624} C_VEL
LIN {X 0,Y 424.872,Z 342.565,A -85,B 0,C 180,E1 -9997.414,E2 -9997.414} C_VEL
LIN {X 0,Y 421.983,Z 342.927,A -85,B 0,C 180,E1 -9998.694,E2 -9998.694} C_VEL
LIN {X 0,Y 419.508,Z 343.232,A -85,B 0,C 180,E1 -9999.728,E2 -9999.728} C_VEL
LIN {X 0,Y 418.424,Z 343.364,A -85,B 0,C 180,E1 -10000.528,E2 -10000.528} C_VEL
LIN {X 0,Y 418.325,Z 343.375,A -85,B 0,C 180,E1 -10000.8,E2 -10000.8} C_VEL
LIN {X 0,Y 418.314,Z 343.378,A -85,B 0,C 180,E1 -10003.604,E2 -10003.604} C_VEL
LIN {X 0,Y 418.314,Z 343.375,A -85,B 0,C 180,E1 -10006.736,E2 -10006.736} C_VEL
LIN {X 0,Y 418.272,Z 343.384,A -85,B 0,C 180,E1 -10009.791,E2 -10009.791} C_VEL
LIN {X 0,Y 418.239,Z 343.387,A -85,B 0,C 180,E1 -10012.736,E2 -10012.736} C_VEL
LIN {X 0,Y 418.272,Z 343.385,A -85,B 0,C 180,E1 -10015.904,E2 -10015.904} C_VEL
LIN {X 0,Y 418.266,Z 343.384,A -85,B 0,C 180,E1 -10019.162,E2 -10019.162} C_VEL
LIN {X 0,Y 418.259,Z 343.383,A -85,B 0,C 180,E1 -10022.844,E2 -10022.844} C_VEL
LIN {X 0,Y 418.247,Z 343.384,A -85,B 0,C 180,E1 -10026.238,E2 -10026.238} C_VEL
LIN {X 0,Y 418.254,Z 343.385,A -85,B 0,C 180,E1 -10029.682,E2 -10029.682} C_VEL
LIN {X 0,Y 418.286,Z 343.381,A -85,B 0,C 180,E1 -10032.33,E2 -10032.33} C_VEL
LIN {X 0,Y 418.253,Z 343.386,A -85,B 0,C 180,E1 -10035.111,E2 -10035.111} C_VEL
LIN {X 0,Y 418.243,Z 343.387,A -85,B 0,C 180,E1 -10037.767,E2 -10037.767} C_VEL
LIN {X 0,Y 418.255,Z 343.384,A -85,B 0,C 180,E1 -10040.62,E2 -10040.62} C_VEL
LIN {X 0,Y 418.246,Z 343.384,A -85,B 0,C 180,E1 -10043.976,E2 -10043.976} C_VEL
LIN {X 0,Y 418.261,Z 343.385,A -85,B 0,C 180,E1 -10047.156,E2 -10047.156} C_VEL
LIN {X 0,Y 418.272,Z 343.384,A -85,B 0,C 180,E1 -10050.896,E2 -10050.896} C_VEL
LIN {X 0,Y 418.275,Z 343.382,A -85,B 0,C 180,E1 -10054.096,E2 -10054.096} C_VEL
LIN {X 0,Y 418.242,Z 343.387,A -85,B 0,C 180,E1 -10057.264,E2 -10057.264} C_VEL
LIN {X 0,Y 418.288,Z 343.38,A -85,B 0,C 180,E1 -10060.365,E2 -10060.365} C_VEL
LIN {X 0,Y 418.322,Z 343.376,A -85,B 0,C 180,E1 -10063.405,E2 -10063.405} C_VEL
LIN {X 0,Y 418.351,Z 343.374,A -85,B 0,C 180,E1 -10066.999,E2 -10066.999} C_VEL
LIN {X 0,Y 418.347,Z 343.374,A -85,B 0,C 180,E1 -10070.329,E2 -10070.329} C_VEL
LIN {X 0,Y 418.499,Z 343.354,A -85,B 0,C 180,E1 -10073.249,E2 -10073.249} C_VEL
LIN {X 0,Y 418.342,Z 343.373,A -85,B 0,C 180,E1 -10075.182,E2 -10075.182} C_VEL
LIN {X 0,Y 418.547,Z 343.348,A -85,B 0,C 180,E1 -10078.076,E2 -10078.076} C_VEL
LIN {X 0,Y 418.677,Z 343.333,A -85,B 0,C 180,E1 -10080,E2 -10080} C_VEL
LIN {X 0,Y 418.515,Z 343.353,A -85,B 0,C 180,E1 -10082.888,E2 -10082.888} C_VEL
LIN {X 0,Y 418.511,Z 343.354,A -85,B 0,C 180,E1 -10085.783,E2 -10085.783} C_VEL
LIN {X 0,Y 418.383,Z 343.372,A -85,B 0,C 180,E1 -10088.696,E2 -10088.696} C_VEL
LIN {X 0,Y 418.32,Z 343.376,A -85,B 0,C 180,E1 -10091.631,E2 -10091.631} C_VEL
LIN {X 0,Y 418.308,Z 343.378,A -85,B 0,C 180,E1 -10094.597,E2 -10094.597} C_VEL
LIN {X 0,Y 418.294,Z 343.38,A -85,B 0,C 180,E1 -10097.604,E2 -10097.604} C_VEL
LIN {X 0,Y 418.256,Z 343.385,A -85,B 0,C 180,E1 -10100.663,E2 -10100.663} C_VEL
LIN {X 0,Y 418.293,Z 343.382,A -85,B 0,C 180,E1 -10103.781,E2 -10103.781} C_VEL
LIN {X 0,Y 418.315,Z 343.377,A -85,B 0,C 180,E1 -10107.07,E2 -10107.07} C_VEL
LIN {X 0,Y 418.249,Z 343.388,A -85,B 0,C 180,E1 -10110.272,E2 -10110.272} C_VEL
LIN {X 0,Y 418.253,Z 343.387,A -85,B 0,C 180,E1 -10113.677,E2 -10113.677} C_VEL
LIN {X 0,Y 418.25,Z 343.386,A -85,B 0,C 180,E1 -10117.223,E2 -10117.223} C_VEL
LIN {X 0,Y 418.256,Z 343.386,A -85,B 0,C 180,E1 -10119.682,E2 -10119.682} C_VEL
LIN {X 0,Y 418.234,Z 343.39,A -85,B 0,C 180,E1 -10122.321,E2 -10122.321} C_VEL
LIN {X 0,Y 418.243,Z 343.388,A -85,B 0,C 180,E1 -10125.109,E2 -10125.109} C_VEL
LIN {X 0,Y 418.277,Z 343.585,A -85,B 0,C 180,E1 -10127.014,E2 -10127.014} C_VEL
LIN {X 0,Y 420.288,Z 353.597,A -85,B 0,C 180,E1 -10130.283,E2 -10130.283} C_VEL
LIN {X 0,Y 421.684,Z 360.743,A -85,B 0,C 180,E1 -10132.531,E2 -10132.531} C_VEL
LIN {X 0,Y 421.809,Z 364.804,A -85,B 0,C 180,E1 -10133.737,E2 -10133.737} C_VEL
LIN {X 0,Y 420.799,Z 376.8,A -85,B 0,C 180,E1 -10137.141,E2 -10137.141} C_VEL
LIN {X 0,Y 420.013,Z 387.922,A -85,B 0,C 180,E1 -10140.229,E2 -10140.229} C_VEL
LIN {X 0,Y 419.236,Z 400.398,A -85,B 0,C 180,E1 -10143.625,E2 -10143.625} C_VEL
LIN {X 0,Y 418.655,Z 412.129,A -85,B 0,C 180,E1 -10146.765,E2 -10146.765} C_VEL
LIN {X 0,Y 418.107,Z 425.706,A -85,B 0,C 180,E1 -10150.355,E2 -10150.355} C_VEL
LIN {X 0,Y 417.788,Z 435.779,A -85,B 0,C 180,E1 -10152.986,E2 -10152.986} C_VEL
LIN {X 0,Y 419.287,Z 451.895,A -85,B 0,C 180,E1 -10153.565,E2 -10153.565} C_VEL
LIN {X 0,Y 420.124,Z 464.896,A -85,B 0,C 180,E1 -10154.228,E2 -10154.228} C_VEL
LIN {X 0,Y 420.477,Z 471.069,A -85,B 0,C 180,E1 -10154.613,E2 -10154.613} C_VEL
LIN {X 0,Y 419.734,Z 482.708,A -85,B 0,C 180,E1 -10155.454,E2 -10155.454} C_VEL
LIN {X 0,Y 419.099,Z 493.35,A -85,B 0,C 180,E1 -10156.422,E2 -10156.422} C_VEL
LIN {X 0,Y 418.576,Z 504.107,A -85,B 0,C 180,E1 -10157.639,E2 -10157.639} C_VEL
LIN {X 0,Y 418.085,Z 512.893,A -85,B 0,C 180,E1 -10158.854,E2 -10158.854} C_VEL
LIN {X 0,Y 417.677,Z 521.472,A -85,B 0,C 180,E1 -10160.313,E2 -10160.313} C_VEL
LIN {X 0,Y 417.568,Z 528.37,A -85,B 0,C 180,E1 -10161.775,E2 -10161.775} C_VEL
LIN {X 0,Y 417.528,Z 533.993,A -85,B 0,C 180,E1 -10163.273,E2 -10163.273} C_VEL
LIN {X 0,Y 417.601,Z 538.116,A -85,B 0,C 180,E1 -10164.689,E2 -10164.689} C_VEL
LIN {X 0,Y 417.672,Z 541.239,A -85,B 0,C 180,E1 -10166.141,E2 -10166.141} C_VEL
LIN {X 0,Y 417.666,Z 542.743,A -85,B 0,C 180,E1 -10167.106,E2 -10167.106} C_VEL
LIN {X 0,Y 417.689,Z 543.782,A -85,B 0,C 180,E1 -10168.071,E2 -10168.071} C_VEL
LIN {X 0,Y 417.785,Z 544.38,A -85,B 0,C 180,E1 -10169.036,E2 -10169.036} C_VEL
LIN {X 0,Y 417.908,Z 544.563,A -85,B 0,C 180,E1 -10170,E2 -10170} C_VEL
LIN {X 0,Y 417.922,Z 544.309,A -85,B 0,C 180,E1 -10170.964,E2 -10170.964} C_VEL
LIN {X 0,Y 417.716,Z 543.553,A -85,B 0,C 180,E1 -10171.928,E2 -10171.928} C_VEL
LIN {X 0,Y 417.706,Z 542.39,A -85,B 0,C 180,E1 -10172.893,E2 -10172.893} C_VEL
LIN {X 0,Y 417.753,Z 539.828,A -85,B 0,C 180,E1 -10174.342,E2 -10174.342} C_VEL
LIN {X 0,Y 417.62,Z 535.137,A -85,B 0,C 180,E1 -10176.149,E2 -10176.149} C_VEL
LIN {X 0,Y 417.595,Z 528.547,A -85,B 0,C 180,E1 -10177.981,E2 -10177.981} C_VEL
LIN {X 0,Y 417.673,Z 521.839,A -85,B 0,C 180,E1 -10179.443,E2 -10179.443} C_VEL
LIN {X 0,Y 417.986,Z 513.612,A -85,B 0,C 180,E1 -10180.904,E2 -10180.904} C_VEL
LIN {X 0,Y 418.527,Z 503.461,A -85,B 0,C 180,E1 -10182.363,E2 -10182.363} C_VEL
LIN {X 0,Y 418.943,Z 494.518,A -85,B 0,C 180,E1 -10183.43,E2 -10183.43} C_VEL
LIN {X 0,Y 419.732,Z 483.252,A -85,B 0,C 180,E1 -10184.546,E2 -10184.546} C_VEL
LIN {X 0,Y 420.612,Z 471.207,A -85,B 0,C 180,E1 -10185.506,E2 -10185.506} C_VEL
LIN {X 0,Y 420.226,Z 457.869,A -85,B 0,C 180,E1 -10186.393,E2 -10186.393} C_VEL
LIN {X 0,Y 419.761,Z 444.525,A -85,B 0,C 180,E1 -10187.088,E2 -10187.088} C_VEL
LIN {X 0,Y 418.094,Z 430.183,A -85,B 0,C 180,E1 -10187.691,E2 -10187.691} C_VEL
LIN {X 0,Y 417.801,Z 427.594,A -85,B 0,C 180,E1 -10187.815,E2 -10187.815} C_VEL
LIN {X 0,Y 418.006,Z 414.01,A -85,B 0,C 180,E1 -10191.191,E2 -10191.191} C_VEL
LIN {X 0,Y 418.383,Z 400.777,A -85,B 0,C 180,E1 -10194.567,E2 -10194.567} C_VEL
LIN {X 0,Y 418.84,Z 387.747,A -85,B 0,C 180,E1 -10198.024,E2 -10198.024} C_VEL
LIN {X 0,Y 419.451,Z 376.07,A -85,B 0,C 180,E1 -10201.293,E2 -10201.293} C_VEL
LIN {X 0,Y 420.337,Z 364.949,A -85,B 0,C 180,E1 -10204.644,E2 -10204.644} C_VEL
LIN {X 0,Y 421.069,Z 358.452,A -85,B 0,C 180,E1 -10206.759,E2 -10206.759} C_VEL
LIN {X 0,Y 420.227,Z 352.988,A -85,B 0,C 180,E1 -10208.841,E2 -10208.841} C_VEL
LIN {X 0,Y 419.01,Z 346.883,A -85,B 0,C 180,E1 -10211.522,E2 -10211.522} C_VEL
LIN {X 0,Y 418.229,Z 343.391,A -85,B 0,C 180,E1 -10213.388,E2 -10213.388} C_VEL
LIN {X 0,Y 418.212,Z 343.391,A -85,B 0,C 180,E1 -10216.449,E2 -10216.449} C_VEL
LIN {X 0,Y 418.226,Z 343.389,A -85,B 0,C 180,E1 -10219.13,E2 -10219.13} C_VEL
LIN {X 0,Y 418.237,Z 343.387,A -85,B 0,C 180,E1 -10222.166,E2 -10222.166} C_VEL
LIN {X 0,Y 418.27,Z 343.383,A -85,B 0,C 180,E1 -10225.42,E2 -10225.42} C_VEL
LIN {X 0,Y 418.215,Z 343.39,A -85,B 0,C 180,E1 -10228.604,E2 -10228.604} C_VEL
LIN {X 0,Y 418.295,Z 343.379,A -85,B 0,C 180,E1 -10231.937,E2 -10231.937} C_VEL
LIN {X 0,Y 418.294,Z 343.381,A -85,B 0,C 180,E1 -10235.163,E2 -10235.163} C_VEL
LIN {X 0,Y 418.238,Z 343.389,A -85,B 0,C 180,E1 -10238.304,E2 -10238.304} C_VEL
LIN {X 0,Y 418.288,Z 343.384,A -85,B 0,C 180,E1 -10241.383,E2 -10241.383} C_VEL
LIN {X 0,Y 418.351,Z 343.566,A -85,B 0,C 180,E1 -10242.029,E2 -10242.029} C_VEL
LIN {X 0,Y 422.259,Z 354.565,A -85,B 0,C 180,E1 -10242.947,E2 -10242.947} C_VEL
LIN {X 0,Y 423.652,Z 359.326,A -85,B 0,C 180,E1 -10243.381,E2 -10243.381} C_VEL
LIN {X 0,Y 423.038,Z 370.926,A -85,B 0,C 180,E1 -10244.338,E2 -10244.338} C_VEL
LIN {X 0,Y 422.267,Z 381.55,A -85,B 0,C 180,E1 -10245.421,E2 -10245.421} C_VEL
LIN {X 0,Y 421.673,Z 390.173,A -85,B 0,C 180,E1 -10246.506,E2 -10246.506} C_VEL
LIN {X 0,Y 420.962,Z 398.109,A -85,B 0,C 180,E1 -10247.71,E2 -10247.71} C_VEL
LIN {X 0,Y 420.281,Z 405.809,A -85,B 0,C 180,E1 -10249.156,E2 -10249.156} C_VEL
LIN {X 0,Y 419.646,Z 412.896,A -85,B 0,C 180,E1 -10250.846,E2 -10250.846} C_VEL
LIN {X 0,Y 419.185,Z 417.57,A -85,B 0,C 180,E1 -10252.292,E2 -10252.292} C_VEL
LIN {X 0,Y 418.827,Z 421.137,A -85,B 0,C 180,E1 -10253.738,E2 -10253.738} C_VEL
LIN {X 0,Y 418.441,Z 423.698,A -85,B 0,C 180,E1 -10255.183,E2 -10255.183} C_VEL
LIN {X 0,Y 418.346,Z 424.831,A -85,B 0,C 180,E1 -10256.147,E2 -10256.147} C_VEL
LIN {X 0,Y 418.215,Z 425.922,A -85,B 0,C 180,E1 -10258.074,E2 -10258.074} C_VEL
LIN {X 0,Y 418.158,Z 425.841,A -85,B 0,C 180,E1 -10259.037,E2 -10259.037} C_VEL
LIN {X 0,Y 418.117,Z 425.364,A -85,B 0,C 180,E1 -10260,E2 -10260} C_VEL
LIN {X 0,Y 418.023,Z 424.51,A -85,B 0,C 180,E1 -10260.963,E2 -10260.963} C_VEL
LIN {X 0,Y 418.109,Z 423.223,A -85,B 0,C 180,E1 -10261.926,E2 -10261.926} C_VEL
LIN {X 0,Y 418.2,Z 420.5,A -85,B 0,C 180,E1 -10263.372,E2 -10263.372} C_VEL
LIN {X 0,Y 418.317,Z 416.77,A -85,B 0,C 180,E1 -10264.819,E2 -10264.819} C_VEL
LIN {X 0,Y 418.648,Z 411.906,A -85,B 0,C 180,E1 -10266.264,E2 -10266.264} C_VEL
LIN {X 0,Y 419.116,Z 405.78,A -85,B 0,C 180,E1 -10267.709,E2 -10267.709} C_VEL
LIN {X 0,Y 419.468,Z 398.214,A -85,B 0,C 180,E1 -10269.158,E2 -10269.158} C_VEL
LIN {X 0,Y 419.844,Z 390.536,A -85,B 0,C 180,E1 -10270.367,E2 -10270.367} C_VEL
LIN {X 0,Y 420.442,Z 381.277,A -85,B 0,C 180,E1 -10271.571,E2 -10271.571} C_VEL
LIN {X 0,Y 420.954,Z 371.062,A -85,B 0,C 180,E1 -10272.658,E2 -10272.658} C_VEL
LIN {X 0,Y 421.38,Z 360.116,A -85,B 0,C 180,E1 -10273.607,E2 -10273.607} C_VEL
LIN {X 0,Y 421.596,Z 355.989,A -85,B 0,C 180,E1 -10273.913,E2 -10273.913} C_VEL
LIN {X 0,Y 418.329,Z 343.376,A -85,B 0,C 180,E1 -10274.845,E2 -10274.845} C_VEL
LIN {X 0,Y 418.283,Z 343.381,A -85,B 0,C 180,E1 -10277.604,E2 -10277.604} C_VEL
LIN {X 0,Y 418.253,Z 343.385,A -85,B 0,C 180,E1 -10280.663,E2 -10280.663} C_VEL
LIN {X 0,Y 418.291,Z 343.381,A -85,B 0,C 180,E1 -10283.781,E2 -10283.781} C_VEL
LIN {X 0,Y 418.313,Z 343.379,A -85,B 0,C 180,E1 -10287.07,E2 -10287.07} C_VEL
LIN {X 0,Y 418.247,Z 343.386,A -85,B 0,C 180,E1 -10290.272,E2 -10290.272} C_VEL
LIN {X 0,Y 418.251,Z 343.384,A -85,B 0,C 180,E1 -10293.677,E2 -10293.677} C_VEL
LIN {X 0,Y 418.249,Z 343.386,A -85,B 0,C 180,E1 -10297.223,E2 -10297.223} C_VEL
LIN {X 0,Y 418.267,Z 343.383,A -85,B 0,C 180,E1 -10299.68,E2 -10299.68} C_VEL
LIN {X 0,Y 418.247,Z 343.388,A -85,B 0,C 180,E1 -10302.323,E2 -10302.323} C_VEL
LIN {X 0,Y 418.242,Z 343.388,A -85,B 0,C 180,E1 -10305.109,E2 -10305.109} C_VEL
LIN {X 0,Y 418.244,Z 343.386,A -85,B 0,C 180,E1 -10307.767,E2 -10307.767} C_VEL
LIN {X 0,Y 418.257,Z 343.387,A -85,B 0,C 180,E1 -10310.619,E2 -10310.619} C_VEL
LIN {X 0,Y 418.244,Z 343.384,A -85,B 0,C 180,E1 -10313.976,E2 -10313.976} C_VEL
LIN {X 0,Y 418.259,Z 343.384,A -85,B 0,C 180,E1 -10317.156,E2 -10317.156} C_VEL
LIN {X 0,Y 418.27,Z 343.384,A -85,B 0,C 180,E1 -10320.895,E2 -10320.895} C_VEL
LIN {X 0,Y 418.272,Z 343.384,A -85,B 0,C 180,E1 -10324.096,E2 -10324.096} C_VEL
LIN {X 0,Y 418.239,Z 343.386,A -85,B 0,C 180,E1 -10327.264,E2 -10327.264} C_VEL
LIN {X 0,Y 418.317,Z 343.381,A -85,B 0,C 180,E1 -10330.366,E2 -10330.366} C_VEL
LIN {X 0,Y 418.318,Z 343.375,A -85,B 0,C 180,E1 -10333.405,E2 -10333.405} C_VEL
LIN {X 0,Y 418.347,Z 343.373,A -85,B 0,C 180,E1 -10336.999,E2 -10336.999} C_VEL
LIN {X 0,Y 418.342,Z 343.375,A -85,B 0,C 180,E1 -10340.329,E2 -10340.329} C_VEL
LIN {X 0,Y 418.488,Z 343.356,A -85,B 0,C 180,E1 -10343.249,E2 -10343.249} C_VEL
LIN {X 0,Y 418.34,Z 343.373,A -85,B 0,C 180,E1 -10345.182,E2 -10345.182} C_VEL
LIN {X 0,Y 418.546,Z 343.353,A -85,B 0,C 180,E1 -10348.076,E2 -10348.076} C_VEL
LIN {X 0,Y 418.672,Z 343.336,A -85,B 0,C 180,E1 -10350,E2 -10350} C_VEL
LIN {X 0,Y 418.512,Z 343.352,A -85,B 0,C 180,E1 -10352.888,E2 -10352.888} C_VEL
LIN {X 0,Y 418.489,Z 343.356,A -85,B 0,C 180,E1 -10356.751,E2 -10356.751} C_VEL
LIN {X 0,Y 418.343,Z 343.375,A -85,B 0,C 180,E1 -10359.671,E2 -10359.671} C_VEL
LIN {X 0,Y 418.325,Z 343.375,A -85,B 0,C 180,E1 -10360.8,E2 -10360.8} C_VEL
LIN {X 0,Y 417.634,Z 343.464,A -85,B 0,C 180,E1 -10361.603,E2 -10361.603} C_VEL
LIN {X 0,Y 414.785,Z 343.816,A -85,B 0,C 180,E1 -10362.909,E2 -10362.909} C_VEL
LIN {X 0,Y 412.382,Z 344.119,A -85,B 0,C 180,E1 -10363.964,E2 -10363.964} C_VEL
LIN {X 0,Y 411.341,Z 344.245,A -85,B 0,C 180,E1 -10364.779,E2 -10364.779} C_VEL
LIN {X 0,Y 411.25,Z 344.255,A -85,B 0,C 180,E1 -10365.055,E2 -10365.055} C_VEL
LIN {X 0,Y 411.254,Z 344.258,A -85,B 0,C 180,E1 -10367.915,E2 -10367.915} C_VEL
LIN {X 0,Y 411.198,Z 344.264,A -85,B 0,C 180,E1 -10371.034,E2 -10371.034} C_VEL
LIN {X 0,Y 411.228,Z 344.261,A -85,B 0,C 180,E1 -10374.216,E2 -10374.216} C_VEL
LIN {X 0,Y 411.26,Z 344.257,A -85,B 0,C 180,E1 -10377.478,E2 -10377.478} C_VEL
LIN {X 0,Y 411.191,Z 344.264,A -85,B 0,C 180,E1 -10380.848,E2 -10380.848} C_VEL
LIN {X 0,Y 411.207,Z 344.26,A -85,B 0,C 180,E1 -10384.334,E2 -10384.334} C_VEL
LIN {X 0,Y 411.197,Z 344.264,A -85,B 0,C 180,E1 -10387.974,E2 -10387.974} C_VEL
LIN {X 0,Y 411.208,Z 344.264,A -85,B 0,C 180,E1 -10391.235,E2 -10391.235} C_VEL
LIN {X 0,Y 411.23,Z 344.26,A -85,B 0,C 180,E1 -10394.484,E2 -10394.484} C_VEL
LIN {X 0,Y 411.18,Z 344.265,A -85,B 0,C 180,E1 -10398.195,E2 -10398.195} C_VEL
LIN {X 0,Y 411.22,Z 344.261,A -85,B 0,C 180,E1 -10400.776,E2 -10400.776} C_VEL
LIN {X 0,Y 411.201,Z 344.263,A -85,B 0,C 180,E1 -10404.472,E2 -10404.472} C_VEL
LIN {X 0,Y 411.21,Z 344.265,A -85,B 0,C 180,E1 -10406.874,E2 -10406.874} C_VEL
LIN {X 0,Y 411.236,Z 344.261,A -85,B 0,C 180,E1 -10410.644,E2 -10410.644} C_VEL
LIN {X 0,Y 411.242,Z 344.259,A -85,B 0,C 180,E1 -10413.62,E2 -10413.62} C_VEL
LIN {X 0,Y 411.207,Z 344.265,A -85,B 0,C 180,E1 -10416.853,E2 -10416.853} C_VEL
LIN {X 0,Y 411.219,Z 344.259,A -85,B 0,C 180,E1 -10420.051,E2 -10420.051} C_VEL
LIN {X 0,Y 411.267,Z 344.255,A -85,B 0,C 180,E1 -10423.131,E2 -10423.131} C_VEL
LIN {X 0,Y 411.31,Z 344.251,A -85,B 0,C 180,E1 -10426.896,E2 -10426.896} C_VEL
LIN {X 0,Y 411.298,Z 344.253,A -85,B 0,C 180,E1 -10430.162,E2 -10430.162} C_VEL
LIN {X 0,Y 411.466,Z 344.231,A -85,B 0,C 180,E1 -10433.133,E2 -10433.133} C_VEL
LIN {X 0,Y 411.313,Z 344.249,A -85,B 0,C 180,E1 -10435.099,E2 -10435.099} C_VEL
LIN {X 0,Y 411.516,Z 344.223,A -85,B 0,C 180,E1 -10438.043,E2 -10438.043} C_VEL
LIN {X 0,Y 411.646,Z 344.208,A -85,B 0,C 180,E1 -10440,E2 -10440} C_VEL
LIN {X 0,Y 411.47,Z 344.231,A -85,B 0,C 180,E1 -10442.937,E2 -10442.937} C_VEL
LIN {X 0,Y 411.472,Z 344.231,A -85,B 0,C 180,E1 -10445.882,E2 -10445.882} C_VEL
LIN {X 0,Y 411.324,Z 344.25,A -85,B 0,C 180,E1 -10448.846,E2 -10448.846} C_VEL
LIN {X 0,Y 411.289,Z 344.252,A -85,B 0,C 180,E1 -10451.833,E2 -10451.833} C_VEL
LIN {X 0,Y 411.265,Z 344.254,A -85,B 0,C 180,E1 -10454.853,E2 -10454.853} C_VEL
LIN {X 0,Y 411.258,Z 344.259,A -85,B 0,C 180,E1 -10457.915,E2 -10457.915} C_VEL
LIN {X 0,Y 411.202,Z 344.263,A -85,B 0,C 180,E1 -10461.034,E2 -10461.034} C_VEL
LIN {X 0,Y 411.232,Z 344.261,A -85,B 0,C 180,E1 -10464.215,E2 -10464.215} C_VEL
LIN {X 0,Y 411.263,Z 344.256,A -85,B 0,C 180,E1 -10467.478,E2 -10467.478} C_VEL
LIN {X 0,Y 411.194,Z 344.262,A -85,B 0,C 180,E1 -10470.847,E2 -10470.847} C_VEL
LIN {X 0,Y 411.211,Z 344.262,A -85,B 0,C 180,E1 -10474.333,E2 -10474.333} C_VEL
LIN {X 0,Y 411.205,Z 344.264,A -85,B 0,C 180,E1 -10477.973,E2 -10477.973} C_VEL
LIN {X 0,Y 411.186,Z 344.266,A -85,B 0,C 180,E1 -10480.504,E2 -10480.504} C_VEL
LIN {X 0,Y 411.177,Z 344.268,A -85,B 0,C 180,E1 -10483.133,E2 -10483.133} C_VEL
LIN {X 0,Y 411.213,Z 344.288,A -85,B 0,C 180,E1 -10486.658,E2 -10486.658} C_VEL
LIN {X 0,Y 413.185,Z 354.129,A -85,B 0,C 180,E1 -10489.945,E2 -10489.945} C_VEL
LIN {X 0,Y 414.817,Z 363.022,A -85,B 0,C 180,E1 -10492.778,E2 -10492.778} C_VEL
LIN {X 0,Y 414.676,Z 367.462,A -85,B 0,C 180,E1 -10494.1,E2 -10494.1} C_VEL
LIN {X 0,Y 413.632,Z 379.769,A -85,B 0,C 180,E1 -10497.642,E2 -10497.642} C_VEL
LIN {X 0,Y 412.793,Z 391.58,A -85,B 0,C 180,E1 -10500.972,E2 -10500.972} C_VEL
LIN {X 0,Y 411.962,Z 405.297,A -85,B 0,C 180,E1 -10504.754,E2 -10504.754} C_VEL
LIN {X 0,Y 411.374,Z 416.944,A -85,B 0,C 180,E1 -10507.923,E2 -10507.923} C_VEL
LIN {X 0,Y 410.889,Z 430.468,A -85,B 0,C 180,E1 -10511.553,E2 -10511.553} C_VEL
LIN {X 0,Y 410.715,Z 435.259,A -85,B 0,C 180,E1 -10512.771,E2 -10512.771} C_VEL
LIN {X 0,Y 412.054,Z 449.837,A -85,B 0,C 180,E1 -10513.291,E2 -10513.291} C_VEL
LIN {X 0,Y 412.945,Z 462.385,A -85,B 0,C 180,E1 -10513.92,E2 -10513.92} C_VEL
LIN {X 0,Y 413.471,Z 471.09,A -85,B 0,C 180,E1 -10514.472,E2 -10514.472} C_VEL
LIN {X 0,Y 412.711,Z 482.51,A -85,B 0,C 180,E1 -10515.327,E2 -10515.327} C_VEL
LIN {X 0,Y 412.038,Z 493.359,A -85,B 0,C 180,E1 -10516.352,E2 -10516.352} C_VEL
LIN {X 0,Y 411.613,Z 502.665,A -85,B 0,C 180,E1 -10517.426,E2 -10517.426} C_VEL
LIN {X 0,Y 411.035,Z 511.512,A -85,B 0,C 180,E1 -10518.66,E2 -10518.66} C_VEL
LIN {X 0,Y 410.644,Z 520.195,A -85,B 0,C 180,E1 -10520.145,E2 -10520.145} C_VEL
LIN {X 0,Y 410.511,Z 527.142,A -85,B 0,C 180,E1 -10521.632,E2 -10521.632} C_VEL
LIN {X 0,Y 410.458,Z 533.169,A -85,B 0,C 180,E1 -10523.265,E2 -10523.265} C_VEL
LIN {X 0,Y 410.556,Z 536.979,A -85,B 0,C 180,E1 -10524.597,E2 -10524.597} C_VEL
LIN {X 0,Y 410.635,Z 540.136,A -85,B 0,C 180,E1 -10526.074,E2 -10526.074} C_VEL
LIN {X 0,Y 410.632,Z 541.653,A -85,B 0,C 180,E1 -10527.057,E2 -10527.057} C_VEL
LIN {X 0,Y 410.658,Z 542.722,A -85,B 0,C 180,E1 -10528.038,E2 -10528.038} C_VEL
LIN {X 0,Y 410.774,Z 543.333,A -85,B 0,C 180,E1 -10529.02,E2 -10529.02} C_VEL
LIN {X 0,Y 410.885,Z 543.523,A -85,B 0,C 180,E1 -10530,E2 -10530} C_VEL
LIN {X 0,Y 410.896,Z 543.275,A -85,B 0,C 180,E1 -10530.98,E2 -10530.98} C_VEL
LIN {X 0,Y 410.678,Z 542.54,A -85,B 0,C 180,E1 -10531.961,E2 -10531.961} C_VEL
LIN {X 0,Y 410.664,Z 541.378,A -85,B 0,C 180,E1 -10532.943,E2 -10532.943} C_VEL
LIN {X 0,Y 410.696,Z 538.827,A -85,B 0,C 180,E1 -10534.416,E2 -10534.416} C_VEL
LIN {X 0,Y 410.539,Z 535.19,A -85,B 0,C 180,E1 -10535.895,E2 -10535.895} C_VEL
LIN {X 0,Y 410.483,Z 530.423,A -85,B 0,C 180,E1 -10537.378,E2 -10537.378} C_VEL
LIN {X 0,Y 410.539,Z 524.42,A -85,B 0,C 180,E1 -10538.863,E2 -10538.863} C_VEL
LIN {X 0,Y 410.707,Z 517.016,A -85,B 0,C 180,E1 -10540.351,E2 -10540.351} C_VEL
LIN {X 0,Y 411.137,Z 507.962,A -85,B 0,C 180,E1 -10541.837,E2 -10541.837} C_VEL
LIN {X 0,Y 411.593,Z 499.625,A -85,B 0,C 180,E1 -10542.975,E2 -10542.975} C_VEL
LIN {X 0,Y 412.454,Z 487.772,A -85,B 0,C 180,E1 -10544.304,E2 -10544.304} C_VEL
LIN {X 0,Y 413.456,Z 475.638,A -85,B 0,C 180,E1 -10545.402,E2 -10545.402} C_VEL
LIN {X 0,Y 413.587,Z 467.497,A -85,B 0,C 180,E1 -10546.03,E2 -10546.03} C_VEL
LIN {X 0,Y 413.366,Z 454.793,A -85,B 0,C 180,E1 -10546.864,E2 -10546.864} C_VEL
LIN {X 0,Y 412.743,Z 442.116,A -85,B 0,C 180,E1 -10547.532,E2 -10547.532} C_VEL
LIN {X 0,Y 410.951,Z 428.231,A -85,B 0,C 180,E1 -10548.146,E2 -10548.146} C_VEL
LIN {X 0,Y 410.749,Z 426.098,A -85,B 0,C 180,E1 -10548.26,E2 -10548.26} C_VEL
LIN {X 0,Y 410.972,Z 413.086,A -85,B 0,C 180,E1 -10551.572,E2 -10551.572} C_VEL
LIN {X 0,Y 411.399,Z 399.539,A -85,B 0,C 180,E1 -10555.121,E2 -10555.121} C_VEL
LIN {X 0,Y 411.893,Z 387.043,A -85,B 0,C 180,E1 -10558.539,E2 -10558.539} C_VEL
LIN {X 0,Y 412.622,Z 375.534,A -85,B 0,C 180,E1 -10561.871,E2 -10561.871} C_VEL
LIN {X 0,Y 413.914,Z 362.873,A -85,B 0,C 180,E1 -10565.858,E2 -10565.858} C_VEL
LIN {X 0,Y 414.137,Z 359.308,A -85,B 0,C 180,E1 -10567.098,E2 -10567.098} C_VEL
LIN {X 0,Y 412.86,Z 352.173,A -85,B 0,C 180,E1 -10570.002,E2 -10570.002} C_VEL
LIN {X 0,Y 411.673,Z 346.456,A -85,B 0,C 180,E1 -10572.77,E2 -10572.77} C_VEL
LIN {X 0,Y 411.162,Z 344.271,A -85,B 0,C 180,E1 -10574.05,E2 -10574.05} C_VEL
LIN {X 0,Y 411.185,Z 344.269,A -85,B 0,C 180,E1 -10577.304,E2 -10577.304} C_VEL
LIN {X 0,Y 411.222,Z 344.261,A -85,B 0,C 180,E1 -10580.776,E2 -10580.776} C_VEL
LIN {X 0,Y 411.203,Z 344.266,A -85,B 0,C 180,E1 -10584.471,E2 -10584.471} C_VEL
LIN {X 0,Y 411.211,Z 344.263,A -85,B 0,C 180,E1 -10586.873,E2 -10586.873} C_VEL
LIN {X 0,Y 411.237,Z 344.259,A -85,B 0,C 180,E1 -10590.644,E2 -10590.644} C_VEL
LIN {X 0,Y 411.241,Z 344.258,A -85,B 0,C 180,E1 -10593.619,E2 -10593.619} C_VEL
LIN {X 0,Y 411.206,Z 344.264,A -85,B 0,C 180,E1 -10596.852,E2 -10596.852} C_VEL
LIN {X 0,Y 411.219,Z 344.264,A -85,B 0,C 180,E1 -10600.05,E2 -10600.05} C_VEL
LIN {X 0,Y 411.271,Z 344.343,A -85,B 0,C 180,E1 -10601.569,E2 -10601.569} C_VEL
LIN {X 0,Y 412.976,Z 348.973,A -85,B 0,C 180,E1 -10601.957,E2 -10601.957} C_VEL
LIN {X 0,Y 416.737,Z 359.944,A -85,B 0,C 180,E1 -10602.967,E2 -10602.967} C_VEL
LIN {X 0,Y 417.124,Z 361.453,A -85,B 0,C 180,E1 -10603.107,E2 -10603.107} C_VEL
LIN {X 0,Y 416.466,Z 372.19,A -85,B 0,C 180,E1 -10604.015,E2 -10604.015} C_VEL
LIN {X 0,Y 415.605,Z 383.114,A -85,B 0,C 180,E1 -10605.161,E2 -10605.161} C_VEL
LIN {X 0,Y 414.957,Z 391.744,A -85,B 0,C 180,E1 -10606.284,E2 -10606.284} C_VEL
LIN {X 0,Y 414.085,Z 400.96,A -85,B 0,C 180,E1 -10607.751,E2 -10607.751} C_VEL
LIN {X 0,Y 413.355,Z 408.372,A -85,B 0,C 180,E1 -10609.221,E2 -10609.221} C_VEL
LIN {X 0,Y 412.758,Z 414.416,A -85,B 0,C 180,E1 -10610.74,E2 -10610.74} C_VEL
LIN {X 0,Y 412.266,Z 418.861,A -85,B 0,C 180,E1 -10612.162,E2 -10612.162} C_VEL
LIN {X 0,Y 411.874,Z 422.36,A -85,B 0,C 180,E1 -10613.632,E2 -10613.632} C_VEL
LIN {X 0,Y 411.46,Z 424.864,A -85,B 0,C 180,E1 -10615.101,E2 -10615.101} C_VEL
LIN {X 0,Y 411.366,Z 425.967,A -85,B 0,C 180,E1 -10616.081,E2 -10616.081} C_VEL
LIN {X 0,Y 411.233,Z 426.694,A -85,B 0,C 180,E1 -10617.061,E2 -10617.061} C_VEL
LIN {X 0,Y 411.214,Z 427.01,A -85,B 0,C 180,E1 -10618.041,E2 -10618.041} C_VEL
LIN {X 0,Y 411.148,Z 426.899,A -85,B 0,C 180,E1 -10619.02,E2 -10619.02} C_VEL
LIN {X 0,Y 411.104,Z 426.392,A -85,B 0,C 180,E1 -10620,E2 -10620} C_VEL
LIN {X 0,Y 410.999,Z 425.509,A -85,B 0,C 180,E1 -10620.98,E2 -10620.98} C_VEL
LIN {X 0,Y 411.086,Z 424.179,A -85,B 0,C 180,E1 -10621.959,E2 -10621.959} C_VEL
LIN {X 0,Y 411.183,Z 421.401,A -85,B 0,C 180,E1 -10623.429,E2 -10623.429} C_VEL
LIN {X 0,Y 411.303,Z 417.608,A -85,B 0,C 180,E1 -10624.901,E2 -10624.901} C_VEL
LIN {X 0,Y 411.655,Z 412.673,A -85,B 0,C 180,E1 -10626.371,E2 -10626.371} C_VEL
LIN {X 0,Y 412.118,Z 406.477,A -85,B 0,C 180,E1 -10627.841,E2 -10627.841} C_VEL
LIN {X 0,Y 412.482,Z 398.832,A -85,B 0,C 180,E1 -10629.315,E2 -10629.315} C_VEL
LIN {X 0,Y 412.887,Z 391.074,A -85,B 0,C 180,E1 -10630.543,E2 -10630.543} C_VEL
LIN {X 0,Y 413.509,Z 381.703,A -85,B 0,C 180,E1 -10631.768,E2 -10631.768} C_VEL
LIN {X 0,Y 414.055,Z 371.371,A -85,B 0,C 180,E1 -10632.872,E2 -10632.872} C_VEL
LIN {X 0,Y 414.473,Z 360.526,A -85,B 0,C 180,E1 -10633.821,E2 -10633.821} C_VEL
LIN {X 0,Y 414.615,Z 357.076,A -85,B 0,C 180,E1 -10634.082,E2 -10634.082} C_VEL
LIN {X 0,Y 411.299,Z 344.253,A -85,B 0,C 180,E1 -10635.041,E2 -10635.041} C_VEL
